    |   movel([0.279628, -1.417351, -2.542506, -0.752532, 1.570796, 1.850424],accel_mss,speed_ms,0,blend_radius_m)
    |   movel([0.279622, -1.416853, -2.542884, -0.752651, 1.570796, 1.850419],accel_mss,speed_ms,0,blend_radius_m)
    |   movel([0.279626, -1.416354, -2.543263, -0.752771, 1.570796, 1.850422],accel_mss,speed_ms,0,blend_radius_m)
    |   movel([0.279638, -1.416064, -2.543483, -0.752841, 1.570796, 1.850434],accel_mss,speed_ms,0,blend_radius_m)
    |   movel([0.279658, -1.415769, -2.543707, -0.752913, 1.570796, 1.850454],accel_mss,speed_ms,0,blend_radius_m)
    |   movel([0.279687, -1.415475, -2.543930, -0.752984, 1.570796, 1.850483],accel_mss,speed_ms,0,blend_radius_m)
    |   movel([0.279726, -1.415198, -2.544139, -0.753051, 1.570796, 1.850522],accel_mss,speed_ms,0,blend_radius_m)
    |   movel([0.279771, -1.414923, -2.544348, -0.753118, 1.570796, 1.850568],accel_mss,speed_ms,0,blend_radius_m)
    |   movel([0.279832, -1.414642, -2.544561, -0.753187, 1.570796, 1.850628],accel_mss,speed_ms,0,blend_radius_m)
    |   movel([0.279917, -1.414283, -2.544832, -0.753274, 1.570796, 1.850713],accel_mss,speed_ms,0,blend_radius_m)
    |   movel([0.280011, -1.413921, -2.545105, -0.753363, 1.570796, 1.850808],accel_mss,speed_ms,0,blend_radius_m)
    |   movel([0.280115, -1.413560, -2.545377, -0.753451, 1.570796, 1.850911],accel_mss,speed_ms,0,blend_radius_m)
    |   movel([0.280391, -1.412635, -2.546075, -0.753679, 1.570796, 1.851188],accel_mss,speed_ms,0,blend_radius_m)
    |   movel([0.280678, -1.411708, -2.546772, -0.753908, 1.570796, 1.851474],accel_mss,speed_ms,0,blend_radius_m)
    |   movel([0.280987, -1.410738, -2.547501, -0.754150, 1.570796, 1.851783],accel_mss,speed_ms,0,blend_radius_m)
    |   movel([0.281302, -1.409763, -2.548232, -0.754394, 1.570796, 1.852098],accel_mss,speed_ms,0,blend_radius_m)
    |   movel([0.281425, -1.409404, -2.548501, -0.754484, 1.570796, 1.852222],accel_mss,speed_ms,0,blend_radius_m)
    |   movel([0.281559, -1.409042, -2.548772, -0.754575, 1.570796, 1.852355],accel_mss,speed_ms,0,blend_radius_m)
    |   movel([0.281701, -1.408680, -2.549042, -0.754667, 1.570796, 1.852497],accel_mss,speed_ms,0,blend_radius_m)
    |   movel([0.281827, -1.408385, -2.549263, -0.754741, 1.570796, 1.852623],accel_mss,speed_ms,0,blend_radius_m)
    |   movel([0.281964, -1.408090, -2.549483, -0.754816, 1.570796, 1.852760],accel_mss,speed_ms,0,blend_radius_m)
    |   movel([0.282113, -1.407794, -2.549704, -0.754891, 1.570796, 1.852909],accel_mss,speed_ms,0,blend_radius_m)
    |   movel([0.282407, -1.407251, -2.550109, -0.755029, 1.570796, 1.853203],accel_mss,speed_ms,0,blend_radius_m)
    |   movel([0.282716, -1.406709, -2.550513, -0.755167, 1.570796, 1.853512],accel_mss,speed_ms,0,blend_radius_m)
    |   movel([0.283060, -1.406138, -2.550938, -0.755314, 1.570796, 1.853856],accel_mss,speed_ms,0,blend_radius_m)
    |   movel([0.283416, -1.405569, -2.551360, -0.755460, 1.570796, 1.854213],accel_mss,speed_ms,0,blend_radius_m)
    |   movel([0.283790, -1.405004, -2.551780, -0.755605, 1.570796, 1.854586],accel_mss,speed_ms,0,blend_radius_m)
    |   movel([0.284177, -1.404442, -2.552197, -0.755751, 1.570796, 1.854973],accel_mss,speed_ms,0,blend_radius_m)
    |   movel([0.284577, -1.403881, -2.552612, -0.755896, 1.570796, 1.855373],accel_mss,speed_ms,0,blend_radius_m)
    |   movel([0.284991, -1.403328, -2.553021, -0.756040, 1.570796, 1.855787],accel_mss,speed_ms,0,blend_radius_m)
    |   movel([0.285421, -1.402776, -2.553429, -0.756184, 1.570796, 1.856217],accel_mss,speed_ms,0,blend_radius_m)
    |   movel([0.285863, -1.402229, -2.553833, -0.756327, 1.570796, 1.856659],accel_mss,speed_ms,0,blend_radius_m)
    |   movel([0.286317, -1.401689, -2.554231, -0.756469, 1.570796, 1.857113],accel_mss,speed_ms,0,blend_radius_m)
    |   movel([0.286768, -1.401172, -2.554612, -0.756605, 1.570796, 1.857565],accel_mss,speed_ms,0,blend_radius_m)
    |   movel([0.287233, -1.400663, -2.554986, -0.756739, 1.570796, 1.858030],accel_mss,speed_ms,0,blend_radius_m)
    |   movel([0.287711, -1.400160, -2.555357, -0.756873, 1.570796, 1.858507],accel_mss,speed_ms,0,blend_radius_m)
    |   movel([0.288202, -1.399665, -2.555720, -0.757004, 1.570796, 1.858998],accel_mss,speed_ms,0,blend_radius_m)
    |   movel([0.288701, -1.399180, -2.556076, -0.757133, 1.570796, 1.859498],accel_mss,speed_ms,0,blend_radius_m)
    |   movel([0.289215, -1.398701, -2.556427, -0.757261, 1.570796, 1.860011],accel_mss,speed_ms,0,blend_radius_m)
    |   movel([0.289741, -1.398229, -2.556773, -0.757387, 1.570796, 1.860537],accel_mss,speed_ms,0,blend_radius_m)
    |   movel([0.290274, -1.397769, -2.557109, -0.757511, 1.570796, 1.861071],accel_mss,speed_ms,0,blend_radius_m)
    |   movel([0.290819, -1.397318, -2.557439, -0.757632, 1.570796, 1.861615],accel_mss,speed_ms,0,blend_radius_m)
    |   movel([0.291362, -1.396889, -2.557752, -0.757748, 1.570796, 1.862158],accel_mss,speed_ms,0,blend_radius_m)
    |   movel([0.291912, -1.396467, -2.558060, -0.757862, 1.570796, 1.862708],accel_mss,speed_ms,0,blend_radius_m)
    |   movel([0.292474, -1.396059, -2.558358, -0.757972, 1.570796, 1.863270],accel_mss,speed_ms,0,blend_radius_m)
    |   movel([0.293042, -1.395660, -2.558648, -0.758080, 1.570796, 1.863838],accel_mss,speed_ms,0,blend_radius_m)
    |   movel([0.293615, -1.395276, -2.558928, -0.758185, 1.570796, 1.864411],accel_mss,speed_ms,0,blend_radius_m)
    |   movel([0.294199, -1.394901, -2.559200, -0.758287, 1.570796, 1.864995],accel_mss,speed_ms,0,blend_radius_m)
    |   movel([0.294788, -1.394541, -2.559462, -0.758385, 1.570796, 1.865584],accel_mss,speed_ms,0,blend_radius_m)
    |   movel([0.295381, -1.394196, -2.559713, -0.758480, 1.570796, 1.866177],accel_mss,speed_ms,0,blend_radius_m)
    |   movel([0.295981, -1.393860, -2.559957, -0.758572, 1.570796, 1.866777],accel_mss,speed_ms,0,blend_radius_m)
    |   movel([0.296585, -1.393541, -2.560188, -0.758660, 1.570796, 1.867381],accel_mss,speed_ms,0,blend_radius_m)
    |   movel([0.297191, -1.393235, -2.560410, -0.758744, 1.570796, 1.867988],accel_mss,speed_ms,0,blend_radius_m)
    |   movel([0.297803, -1.392943, -2.560622, -0.758824, 1.570796, 1.868599],accel_mss,speed_ms,0,blend_radius_m)
    |   movel([0.298417, -1.392666, -2.560822, -0.758901, 1.570796, 1.869213],accel_mss,speed_ms,0,blend_radius_m)
    |   movel([0.299033, -1.392405, -2.561012, -0.758973, 1.570796, 1.869829],accel_mss,speed_ms,0,blend_radius_m)
    |   movel([0.299650, -1.392160, -2.561188, -0.759041, 1.570796, 1.870446],accel_mss,speed_ms,0,blend_radius_m)
    |   movel([0.300268, -1.391928, -2.561356, -0.759105, 1.570796, 1.871064],accel_mss,speed_ms,0,blend_radius_m)
    |   movel([0.300887, -1.391714, -2.561511, -0.759164, 1.570796, 1.871684],accel_mss,speed_ms,0,blend_radius_m)
    |   movel([0.301504, -1.391515, -2.561655, -0.759219, 1.570796, 1.872301],accel_mss,speed_ms,0,blend_radius_m)
    |   movel([0.302008, -1.391368, -2.561761, -0.759260, 1.570796, 1.872804],accel_mss,speed_ms,0,blend_radius_m)
    |   movel([0.302511, -1.391237, -2.561856, -0.759297, 1.570796, 1.873307],accel_mss,speed_ms,0,blend_radius_m)
    |   movel([0.303009, -1.391121, -2.561939, -0.759329, 1.570796, 1.873805],accel_mss,speed_ms,0,blend_radius_m)
    |   movel([0.303506, -1.391023, -2.562010, -0.759356, 1.570796, 1.874302],accel_mss,speed_ms,0,blend_radius_m)
    |   movel([0.304074, -1.390924, -2.562081, -0.759384, 1.570796, 1.874870],accel_mss,speed_ms,0,blend_radius_m)
    |   movel([0.304640, -1.390839, -2.562142, -0.759407, 1.570796, 1.875436],accel_mss,speed_ms,0,blend_radius_m)
    |   movel([0.305199, -1.390768, -2.562194, -0.759427, 1.570796, 1.875995],accel_mss,speed_ms,0,blend_radius_m)
    |   movel([0.305757, -1.390708, -2.562237, -0.759444, 1.570796, 1.876553],accel_mss,speed_ms,0,blend_radius_m)
    |   movel([0.306310, -1.390661, -2.562271, -0.759457, 1.570796, 1.877106],accel_mss,speed_ms,0,blend_radius_m)
    |   movel([0.306859, -1.390626, -2.562296, -0.759467, 1.570796, 1.877656],accel_mss,speed_ms,0,blend_radius_m)
    |   movel([0.307404, -1.390604, -2.562312, -0.759473, 1.570796, 1.878200],accel_mss,speed_ms,0,blend_radius_m)
    |   movel([0.307942, -1.390597, -2.562317, -0.759475, 1.570796, 1.878738],accel_mss,speed_ms,0,blend_radius_m)
    |   movel([0.308401, -1.390603, -2.562313, -0.759473, 1.570796, 1.879198],accel_mss,speed_ms,0,blend_radius_m)
    |   movel([0.308855, -1.390628, -2.562295, -0.759466, 1.570796, 1.879651],accel_mss,speed_ms,0,blend_radius_m)
    |   movel([0.309299, -1.390668, -2.562266, -0.759455, 1.570796, 1.880095],accel_mss,speed_ms,0,blend_radius_m)
    |   movel([0.309734, -1.390725, -2.562225, -0.759439, 1.570796, 1.880531],accel_mss,speed_ms,0,blend_radius_m)
    |   movel([0.310264, -1.390816, -2.562159, -0.759414, 1.570796, 1.881060],accel_mss,speed_ms,0,blend_radius_m)
    |   movel([0.310782, -1.390924, -2.562081, -0.759384, 1.570796, 1.881579],accel_mss,speed_ms,0,blend_radius_m)
    |   movel([0.311288, -1.391050, -2.561990, -0.759349, 1.570796, 1.882084],accel_mss,speed_ms,0,blend_radius_m)
    |   movel([0.311782, -1.391195, -2.561885, -0.759308, 1.570796, 1.882578],accel_mss,speed_ms,0,blend_radius_m)
    |   movel([0.312265, -1.391354, -2.561771, -0.759264, 1.570796, 1.883061],accel_mss,speed_ms,0,blend_radius_m)
    |   movel([0.312730, -1.391535, -2.561640, -0.759214, 1.570796, 1.883527],accel_mss,speed_ms,0,blend_radius_m)
    |   movel([0.313189, -1.391729, -2.561500, -0.759160, 1.570796, 1.883985],accel_mss,speed_ms,0,blend_radius_m)
    |   movel([0.313630, -1.391942, -2.561346, -0.759101, 1.570796, 1.884426],accel_mss,speed_ms,0,blend_radius_m)
    |   movel([0.314058, -1.392169, -2.561182, -0.759038, 1.570796, 1.884854],accel_mss,speed_ms,0,blend_radius_m)
    |   movel([0.314471, -1.392415, -2.561004, -0.758970, 1.570796, 1.885267],accel_mss,speed_ms,0,blend_radius_m)
    |   movel([0.314869, -1.392675, -2.560816, -0.758898, 1.570796, 1.885665],accel_mss,speed_ms,0,blend_radius_m)
    |   movel([0.315252, -1.392952, -2.560615, -0.758822, 1.570796, 1.886049],accel_mss,speed_ms,0,blend_radius_m)
    |   movel([0.315618, -1.393246, -2.560403, -0.758741, 1.570796, 1.886415],accel_mss,speed_ms,0,blend_radius_m)
    |   movel([0.315972, -1.393553, -2.560180, -0.758656, 1.570796, 1.886768],accel_mss,speed_ms,0,blend_radius_m)
    |   movel([0.316307, -1.393875, -2.559946, -0.758568, 1.570796, 1.887103],accel_mss,speed_ms,0,blend_radius_m)
    |   movel([0.316625, -1.394212, -2.559702, -0.758476, 1.570796, 1.887421],accel_mss,speed_ms,0,blend_radius_m)
    |   movel([0.316927, -1.394562, -2.559447, -0.758380, 1.570796, 1.887723],accel_mss,speed_ms,0,blend_radius_m)
    |   movel([0.317209, -1.394927, -2.559182, -0.758280, 1.570796, 1.888006],accel_mss,speed_ms,0,blend_radius_m)
    |   movel([0.317478, -1.395307, -2.558906, -0.758177, 1.570796, 1.888274],accel_mss,speed_ms,0,blend_radius_m)
    |   movel([0.317727, -1.395700, -2.558619, -0.758070, 1.570796, 1.888523],accel_mss,speed_ms,0,blend_radius_m)
    |   movel([0.317959, -1.396104, -2.558325, -0.757960, 1.570796, 1.888756],accel_mss,speed_ms,0,blend_radius_m)
    |   movel([0.318170, -1.396522, -2.558020, -0.757847, 1.570796, 1.888966],accel_mss,speed_ms,0,blend_radius_m)
    |   movel([0.318366, -1.396949, -2.557708, -0.757731, 1.570796, 1.889162],accel_mss,speed_ms,0,blend_radius_m)
    |   movel([0.318541, -1.397389, -2.557387, -0.757613, 1.570796, 1.889338],accel_mss,speed_ms,0,blend_radius_m)
    |   movel([0.318684, -1.397780, -2.557101, -0.757508, 1.570796, 1.889480],accel_mss,speed_ms,0,blend_radius_m)
    |   movel([0.318813, -1.398180, -2.556808, -0.757400, 1.570796, 1.889610],accel_mss,speed_ms,0,blend_radius_m)
    |   movel([0.318930, -1.398586, -2.556511, -0.757292, 1.570796, 1.889726],accel_mss,speed_ms,0,blend_radius_m)
    |   movel([0.319035, -1.398997, -2.556210, -0.757182, 1.570796, 1.889832],accel_mss,speed_ms,0,blend_radius_m)
    |   movel([0.319122, -1.399383, -2.555927, -0.757079, 1.570796, 1.889918],accel_mss,speed_ms,0,blend_radius_m)
    |   movel([0.319192, -1.399776, -2.555638, -0.756974, 1.570796, 1.889989],accel_mss,speed_ms,0,blend_radius_m)
    |   movel([0.319252, -1.400175, -2.555345, -0.756868, 1.570796, 1.890048],accel_mss,speed_ms,0,blend_radius_m)
    |   movel([0.319295, -1.400581, -2.555047, -0.756761, 1.570796, 1.890091],accel_mss,speed_ms,0,blend_radius_m)
    |   movel([0.319326, -1.401001, -2.554738, -0.756650, 1.570796, 1.890123],accel_mss,speed_ms,0,blend_radius_m)
    |   movel([0.319344, -1.401428, -2.554424, -0.756537, 1.570796, 1.890140],accel_mss,speed_ms,0,blend_radius_m)
    |   movel([0.319347, -1.401858, -2.554107, -0.756424, 1.570796, 1.890143],accel_mss,speed_ms,0,blend_radius_m)
    |   movel([0.319338, -1.402295, -2.553784, -0.756310, 1.570796, 1.890134],accel_mss,speed_ms,0,blend_radius_m)
    |   movel([0.319303, -1.402955, -2.553297, -0.756137, 1.570796, 1.890099],accel_mss,speed_ms,0,blend_radius_m)
    |   movel([0.319250, -1.403620, -2.552805, -0.755964, 1.570796, 1.890046],accel_mss,speed_ms,0,blend_radius_m)
    |   movel([0.319177, -1.404290, -2.552309, -0.755790, 1.570796, 1.889973],accel_mss,speed_ms,0,blend_radius_m)
    |   movel([0.319122, -1.404672, -2.552026, -0.755691, 1.570796, 1.889918],accel_mss,speed_ms,0,blend_radius_m)
    |   movel([0.319055, -1.405054, -2.551743, -0.755592, 1.570796, 1.889852],accel_mss,speed_ms,0,blend_radius_m)
    |   movel([0.318973, -1.405442, -2.551455, -0.755492, 1.570796, 1.889770],accel_mss,speed_ms,0,blend_radius_m)
    |   movel([0.318880, -1.405830, -2.551166, -0.755393, 1.570796, 1.889676],accel_mss,speed_ms,0,blend_radius_m)
    |   movel([0.318769, -1.406222, -2.550875, -0.755292, 1.570796, 1.889566],accel_mss,speed_ms,0,blend_radius_m)
    |   movel([0.318582, -1.406841, -2.550414, -0.755134, 1.570796, 1.889378],accel_mss,speed_ms,0,blend_radius_m)
    |   movel([0.318379, -1.407463, -2.549951, -0.754975, 1.570796, 1.889176],accel_mss,speed_ms,0,blend_radius_m)
    |   movel([0.318164, -1.408086, -2.549486, -0.754817, 1.570796, 1.888960],accel_mss,speed_ms,0,blend_radius_m)
    |   movel([0.317935, -1.408706, -2.549023, -0.754660, 1.570796, 1.888732],accel_mss,speed_ms,0,blend_radius_m)
    |   movel([0.317694, -1.409332, -2.548555, -0.754502, 1.570796, 1.888490],accel_mss,speed_ms,0,blend_radius_m)
    |   movel([0.317439, -1.409957, -2.548086, -0.754345, 1.570796, 1.888236],accel_mss,speed_ms,0,blend_radius_m)
    |   movel([0.317172, -1.410581, -2.547619, -0.754189, 1.570796, 1.887968],accel_mss,speed_ms,0,blend_radius_m)
    |   movel([0.316891, -1.411206, -2.547150, -0.754033, 1.570796, 1.887688],accel_mss,speed_ms,0,blend_radius_m)
    |   movel([0.316702, -1.411607, -2.546849, -0.753934, 1.570796, 1.887499],accel_mss,speed_ms,0,blend_radius_m)
    |   movel([0.316500, -1.412006, -2.546548, -0.753834, 1.570796, 1.887297],accel_mss,speed_ms,0,blend_radius_m)
    |   movel([0.316286, -1.412404, -2.546249, -0.753736, 1.570796, 1.887082],accel_mss,speed_ms,0,blend_radius_m)
    |   movel([0.316060, -1.412801, -2.545950, -0.753638, 1.570796, 1.886857],accel_mss,speed_ms,0,blend_radius_m)
    |   movel([0.315822, -1.413196, -2.545652, -0.753541, 1.570796, 1.886618],accel_mss,speed_ms,0,blend_radius_m)
    |   movel([0.315491, -1.413724, -2.545254, -0.753411, 1.570796, 1.886288],accel_mss,speed_ms,0,blend_radius_m)
    |   movel([0.315149, -1.414246, -2.544860, -0.753283, 1.570796, 1.885946],accel_mss,speed_ms,0,blend_radius_m)
    |   movel([0.314795, -1.414766, -2.544466, -0.753156, 1.570796, 1.885591],accel_mss,speed_ms,0,blend_radius_m)
    |   movel([0.314428, -1.415283, -2.544075, -0.753031, 1.570796, 1.885224],accel_mss,speed_ms,0,blend_radius_m)
    |   movel([0.314052, -1.415796, -2.543687, -0.752906, 1.570796, 1.884848],accel_mss,speed_ms,0,blend_radius_m)
    |   speed_ms = 0.003
    |   movel([0.314052, -1.418980, -2.545116, -0.748292, 1.570796, 1.884848],accel_mss,speed_ms,0,blend_radius_m)
    |   speed_ms = 0.007
    |   movel([0.313677, -1.419471, -2.544743, -0.748176, 1.570796, 1.884473],accel_mss,speed_ms,0,blend_radius_m)
    |   movel([0.313291, -1.419955, -2.544373, -0.748061, 1.570796, 1.884087],accel_mss,speed_ms,0,blend_radius_m)
    |   movel([0.312894, -1.420434, -2.544007, -0.747947, 1.570796, 1.883690],accel_mss,speed_ms,0,blend_radius_m)
    |   movel([0.312488, -1.420907, -2.543646, -0.747836, 1.570796, 1.883284],accel_mss,speed_ms,0,blend_radius_m)
    |   movel([0.312070, -1.421375, -2.543288, -0.747726, 1.570796, 1.882867],accel_mss,speed_ms,0,blend_radius_m)
    |   movel([0.311650, -1.421828, -2.542941, -0.747620, 1.570796, 1.882446],accel_mss,speed_ms,0,blend_radius_m)
    |   movel([0.311220, -1.422275, -2.542599, -0.747515, 1.570796, 1.882017],accel_mss,speed_ms,0,blend_radius_m)
    |   movel([0.310783, -1.422715, -2.542262, -0.747413, 1.570796, 1.881579],accel_mss,speed_ms,0,blend_radius_m)
    |   movel([0.310335, -1.423146, -2.541930, -0.747312, 1.570796, 1.881131],accel_mss,speed_ms,0,blend_radius_m)
    |   movel([0.309878, -1.423572, -2.541603, -0.747214, 1.570796, 1.880674],accel_mss,speed_ms,0,blend_radius_m)
    |   movel([0.309414, -1.423989, -2.541283, -0.747117, 1.570796, 1.880210],accel_mss,speed_ms,0,blend_radius_m)
    |   movel([0.308942, -1.424397, -2.540969, -0.747023, 1.570796, 1.879738],accel_mss,speed_ms,0,blend_radius_m)
    |   movel([0.308461, -1.424798, -2.540660, -0.746931, 1.570796, 1.879258],accel_mss,speed_ms,0,blend_radius_m)
    |   movel([0.307976, -1.425188, -2.540359, -0.746842, 1.570796, 1.878772],accel_mss,speed_ms,0,blend_radius_m)
    |   movel([0.307480, -1.425572, -2.540063, -0.746754, 1.570796, 1.878276],accel_mss,speed_ms,0,blend_radius_m)
    |   movel([0.307008, -1.425924, -2.539791, -0.746674, 1.570796, 1.877805],accel_mss,speed_ms,0,blend_radius_m)
    |   movel([0.306532, -1.426271, -2.539524, -0.746595, 1.570796, 1.877329],accel_mss,speed_ms,0,blend_radius_m)
    |   movel([0.306049, -1.426607, -2.539263, -0.746518, 1.570796, 1.876845],accel_mss,speed_ms,0,blend_radius_m)
    |   movel([0.305564, -1.426936, -2.539009, -0.746444, 1.570796, 1.876360],accel_mss,speed_ms,0,blend_radius_m)
    |   movel([0.305072, -1.427259, -2.538759, -0.746371, 1.570796, 1.875869],accel_mss,speed_ms,0,blend_radius_m)
    |   movel([0.304596, -1.427558, -2.538528, -0.746303, 1.570796, 1.875392],accel_mss,speed_ms,0,blend_radius_m)
    |   movel([0.304118, -1.427847, -2.538304, -0.746238, 1.570796, 1.874915],accel_mss,speed_ms,0,blend_radius_m)
    |   movel([0.303635, -1.428129, -2.538085, -0.746175, 1.570796, 1.874431],accel_mss,speed_ms,0,blend_radius_m)
    |   movel([0.303149, -1.428400, -2.537875, -0.746114, 1.570796, 1.873945],accel_mss,speed_ms,0,blend_radius_m)
    |   movel([0.302659, -1.428662, -2.537672, -0.746055, 1.570796, 1.873456],accel_mss,speed_ms,0,blend_radius_m)
    |   movel([0.302165, -1.428914, -2.537476, -0.745999, 1.570796, 1.872961],accel_mss,speed_ms,0,blend_radius_m)
    |   movel([0.301669, -1.429155, -2.537289, -0.745945, 1.570796, 1.872465],accel_mss,speed_ms,0,blend_radius_m)
    |   movel([0.301171, -1.429387, -2.537108, -0.745893, 1.570796, 1.871967],accel_mss,speed_ms,0,blend_radius_m)
    |   movel([0.300669, -1.429609, -2.536936, -0.745844, 1.570796, 1.871465],accel_mss,speed_ms,0,blend_radius_m)
    |   movel([0.300169, -1.429819, -2.536773, -0.745797, 1.570796, 1.870966],accel_mss,speed_ms,0,blend_radius_m)
    |   movel([0.299643, -1.430029, -2.536609, -0.745751, 1.570796, 1.870440],accel_mss,speed_ms,0,blend_radius_m)
    |   movel([0.299116, -1.430229, -2.536454, -0.745706, 1.570796, 1.869913],accel_mss,speed_ms,0,blend_radius_m)
    |   movel([0.298589, -1.430419, -2.536306, -0.745664, 1.570796, 1.869385],accel_mss,speed_ms,0,blend_radius_m)
    |   movel([0.298060, -1.430599, -2.536165, -0.745625, 1.570796, 1.868856],accel_mss,speed_ms,0,blend_radius_m)
    |   movel([0.297533, -1.430769, -2.536033, -0.745587, 1.570796, 1.868329],accel_mss,speed_ms,0,blend_radius_m)
    |   movel([0.297159, -1.430881, -2.535946, -0.745562, 1.570796, 1.867955],accel_mss,speed_ms,0,blend_radius_m)
    |   movel([0.296785, -1.430981, -2.535868, -0.745540, 1.570796, 1.867581],accel_mss,speed_ms,0,blend_radius_m)
    |   movel([0.296415, -1.431068, -2.535800, -0.745521, 1.570796, 1.867211],accel_mss,speed_ms,0,blend_radius_m)
    |   movel([0.296044, -1.431146, -2.535739, -0.745504, 1.570796, 1.866840],accel_mss,speed_ms,0,blend_radius_m)
    |   movel([0.295677, -1.431211, -2.535688, -0.745490, 1.570796, 1.866474],accel_mss,speed_ms,0,blend_radius_m)
    |   movel([0.295078, -1.431301, -2.535618, -0.745470, 1.570796, 1.865874],accel_mss,speed_ms,0,blend_radius_m)
    |   movel([0.294481, -1.431382, -2.535555, -0.745452, 1.570796, 1.865278],accel_mss,speed_ms,0,blend_radius_m)
    |   movel([0.293889, -1.431452, -2.535500, -0.745437, 1.570796, 1.864685],accel_mss,speed_ms,0,blend_radius_m)
    |   movel([0.293298, -1.431509, -2.535456, -0.745424, 1.570796, 1.864095],accel_mss,speed_ms,0,blend_radius_m)
    |   movel([0.292712, -1.431558, -2.535417, -0.745413, 1.570796, 1.863509],accel_mss,speed_ms,0,blend_radius_m)
    |   movel([0.292131, -1.431595, -2.535388, -0.745405, 1.570796, 1.862927],accel_mss,speed_ms,0,blend_radius_m)
    |   movel([0.291553, -1.431620, -2.535369, -0.745400, 1.570796, 1.862349],accel_mss,speed_ms,0,blend_radius_m)
    |   movel([0.290978, -1.431636, -2.535356, -0.745396, 1.570796, 1.861774],accel_mss,speed_ms,0,blend_radius_m)
    |   movel([0.290633, -1.431636, -2.535357, -0.745396, 1.570796, 1.861429],accel_mss,speed_ms,0,blend_radius_m)
    |   movel([0.290291, -1.431623, -2.535367, -0.745399, 1.570796, 1.861088],accel_mss,speed_ms,0,blend_radius_m)
    |   movel([0.289956, -1.431600, -2.535385, -0.745404, 1.570796, 1.860752],accel_mss,speed_ms,0,blend_radius_m)
    |   movel([0.289629, -1.431563, -2.535413, -0.745412, 1.570796, 1.860425],accel_mss,speed_ms,0,blend_radius_m)
    |   movel([0.289306, -1.431515, -2.535451, -0.745423, 1.570796, 1.860102],accel_mss,speed_ms,0,blend_radius_m)
    |   movel([0.288849, -1.431430, -2.535517, -0.745442, 1.570796, 1.859645],accel_mss,speed_ms,0,blend_radius_m)
    |   movel([0.288400, -1.431335, -2.535592, -0.745462, 1.570796, 1.859196],accel_mss,speed_ms,0,blend_radius_m)
    |   movel([0.287956, -1.431229, -2.535674, -0.745486, 1.570796, 1.858752],accel_mss,speed_ms,0,blend_radius_m)
    |   movel([0.287522, -1.431112, -2.535765, -0.745511, 1.570796, 1.858319],accel_mss,speed_ms,0,blend_radius_m)
    |   movel([0.287095, -1.430983, -2.535866, -0.745540, 1.570796, 1.857891],accel_mss,speed_ms,0,blend_radius_m)
    |   movel([0.286701, -1.430853, -2.535968, -0.745569, 1.570796, 1.857497],accel_mss,speed_ms,0,blend_radius_m)
    |   movel([0.286315, -1.430708, -2.536081, -0.745601, 1.570796, 1.857112],accel_mss,speed_ms,0,blend_radius_m)
    |   movel([0.285940, -1.430552, -2.536202, -0.745635, 1.570796, 1.856736],accel_mss,speed_ms,0,blend_radius_m)
    |   movel([0.285575, -1.430384, -2.536333, -0.745672, 1.570796, 1.856371],accel_mss,speed_ms,0,blend_radius_m)
    |   movel([0.285220, -1.430204, -2.536473, -0.745712, 1.570796, 1.856016],accel_mss,speed_ms,0,blend_radius_m)
    |   movel([0.284876, -1.430011, -2.536623, -0.745755, 1.570796, 1.855672],accel_mss,speed_ms,0,blend_radius_m)
    |   movel([0.284542, -1.429806, -2.536782, -0.745800, 1.570796, 1.855338],accel_mss,speed_ms,0,blend_radius_m)
    |   movel([0.284217, -1.429591, -2.536950, -0.745848, 1.570796, 1.855014],accel_mss,speed_ms,0,blend_radius_m)
    |   movel([0.283905, -1.429364, -2.537126, -0.745898, 1.570796, 1.854702],accel_mss,speed_ms,0,blend_radius_m)
    |   movel([0.283606, -1.429126, -2.537311, -0.745951, 1.570796, 1.854402],accel_mss,speed_ms,0,blend_radius_m)
    |   movel([0.283296, -1.428863, -2.537516, -0.746010, 1.570796, 1.854092],accel_mss,speed_ms,0,blend_radius_m)
    |   movel([0.282998, -1.428590, -2.537728, -0.746071, 1.570796, 1.853794],accel_mss,speed_ms,0,blend_radius_m)
    |   movel([0.282710, -1.428306, -2.537948, -0.746135, 1.570796, 1.853506],accel_mss,speed_ms,0,blend_radius_m)
    |   movel([0.282433, -1.428013, -2.538175, -0.746201, 1.570796, 1.853230],accel_mss,speed_ms,0,blend_radius_m)
    |   movel([0.282168, -1.427713, -2.538408, -0.746268, 1.570796, 1.852964],accel_mss,speed_ms,0,blend_radius_m)
    |   movel([0.281908, -1.427391, -2.538657, -0.746341, 1.570796, 1.852705],accel_mss,speed_ms,0,blend_radius_m)
    |   movel([0.281660, -1.427063, -2.538911, -0.746415, 1.570796, 1.852456],accel_mss,speed_ms,0,blend_radius_m)
    |   movel([0.281424, -1.426723, -2.539174, -0.746492, 1.570796, 1.852220],accel_mss,speed_ms,0,blend_radius_m)
    |   movel([0.281204, -1.426373, -2.539445, -0.746571, 1.570796, 1.852000],accel_mss,speed_ms,0,blend_radius_m)
    |   movel([0.280995, -1.426015, -2.539721, -0.746653, 1.570796, 1.851791],accel_mss,speed_ms,0,blend_radius_m)
    |   movel([0.280805, -1.425654, -2.540000, -0.746735, 1.570796, 1.851601],accel_mss,speed_ms,0,blend_radius_m)
    |   movel([0.280628, -1.425285, -2.540285, -0.746819, 1.570796, 1.851424],accel_mss,speed_ms,0,blend_radius_m)
    |   movel([0.280467, -1.424906, -2.540577, -0.746906, 1.570796, 1.851263],accel_mss,speed_ms,0,blend_radius_m)
    |   movel([0.280320, -1.424517, -2.540876, -0.746996, 1.570796, 1.851116],accel_mss,speed_ms,0,blend_radius_m)
    |   movel([0.280187, -1.424121, -2.541181, -0.747087, 1.570796, 1.850983],accel_mss,speed_ms,0,blend_radius_m)
    |   movel([0.280067, -1.423708, -2.541499, -0.747182, 1.570796, 1.850863],accel_mss,speed_ms,0,blend_radius_m)
    |   movel([0.279961, -1.423286, -2.541823, -0.747280, 1.570796, 1.850757],accel_mss,speed_ms,0,blend_radius_m)
    |   movel([0.279870, -1.422858, -2.542152, -0.747379, 1.570796, 1.850667],accel_mss,speed_ms,0,blend_radius_m)
    |   movel([0.279795, -1.422422, -2.542486, -0.747481, 1.570796, 1.850592],accel_mss,speed_ms,0,blend_radius_m)
    |   movel([0.279735, -1.421980, -2.542825, -0.747584, 1.570796, 1.850532],accel_mss,speed_ms,0,blend_radius_m)
    |   movel([0.279686, -1.421501, -2.543192, -0.747696, 1.570796, 1.850483],accel_mss,speed_ms,0,blend_radius_m)
    |   movel([0.279652, -1.421019, -2.543561, -0.747810, 1.570796, 1.850448],accel_mss,speed_ms,0,blend_radius_m)
    |   movel([0.279628, -1.420531, -2.543934, -0.747925, 1.570796, 1.850424],accel_mss,speed_ms,0,blend_radius_m)
    |   movel([0.279622, -1.420035, -2.544313, -0.748042, 1.570796, 1.850419],accel_mss,speed_ms,0,blend_radius_m)
    |   movel([0.279626, -1.419537, -2.544692, -0.748160, 1.570796, 1.850422],accel_mss,speed_ms,0,blend_radius_m)
    |   movel([0.279638, -1.419248, -2.544913, -0.748229, 1.570796, 1.850434],accel_mss,speed_ms,0,blend_radius_m)
    |   movel([0.279658, -1.418954, -2.545137, -0.748299, 1.570796, 1.850454],accel_mss,speed_ms,0,blend_radius_m)
    |   movel([0.279687, -1.418660, -2.545360, -0.748369, 1.570796, 1.850483],accel_mss,speed_ms,0,blend_radius_m)
    |   movel([0.279726, -1.418384, -2.545570, -0.748435, 1.570796, 1.850522],accel_mss,speed_ms,0,blend_radius_m)
    |   movel([0.279771, -1.418110, -2.545779, -0.748500, 1.570796, 1.850568],accel_mss,speed_ms,0,blend_radius_m)
    |   movel([0.279832, -1.417829, -2.545992, -0.748568, 1.570796, 1.850628],accel_mss,speed_ms,0,blend_radius_m)
    |   movel([0.279917, -1.417472, -2.546264, -0.748654, 1.570796, 1.850713],accel_mss,speed_ms,0,blend_radius_m)
    |   movel([0.280011, -1.417111, -2.546538, -0.748740, 1.570796, 1.850808],accel_mss,speed_ms,0,blend_radius_m)
    |   movel([0.280115, -1.416751, -2.546811, -0.748827, 1.570796, 1.850911],accel_mss,speed_ms,0,blend_radius_m)
    |   movel([0.280391, -1.415829, -2.547509, -0.749051, 1.570796, 1.851188],accel_mss,speed_ms,0,blend_radius_m)
    |   movel([0.280678, -1.414904, -2.548209, -0.749276, 1.570796, 1.851474],accel_mss,speed_ms,0,blend_radius_m)
    |   movel([0.280987, -1.413936, -2.548939, -0.749513, 1.570796, 1.851783],accel_mss,speed_ms,0,blend_radius_m)
    |   movel([0.281302, -1.412965, -2.549671, -0.749753, 1.570796, 1.852098],accel_mss,speed_ms,0,blend_radius_m)
    |   movel([0.281425, -1.412607, -2.549941, -0.749842, 1.570796, 1.852222],accel_mss,speed_ms,0,blend_radius_m)
    |   movel([0.281559, -1.412245, -2.550213, -0.749931, 1.570796, 1.852355],accel_mss,speed_ms,0,blend_radius_m)
    |   movel([0.281701, -1.411885, -2.550483, -0.750021, 1.570796, 1.852497],accel_mss,speed_ms,0,blend_radius_m)
    |   movel([0.281827, -1.411590, -2.550704, -0.750094, 1.570796, 1.852623],accel_mss,speed_ms,0,blend_radius_m)
    |   movel([0.281964, -1.411296, -2.550925, -0.750168, 1.570796, 1.852760],accel_mss,speed_ms,0,blend_radius_m)
    |   movel([0.282113, -1.411001, -2.551146, -0.750241, 1.570796, 1.852909],accel_mss,speed_ms,0,blend_radius_m)
    |   movel([0.282407, -1.410459, -2.551553, -0.750377, 1.570796, 1.853203],accel_mss,speed_ms,0,blend_radius_m)
    |   movel([0.282716, -1.409919, -2.551957, -0.750513, 1.570796, 1.853512],accel_mss,speed_ms,0,blend_radius_m)
    |   movel([0.283060, -1.409349, -2.552383, -0.750657, 1.570796, 1.853856],accel_mss,speed_ms,0,blend_radius_m)
    |   movel([0.283416, -1.408782, -2.552807, -0.750800, 1.570796, 1.854213],accel_mss,speed_ms,0,blend_radius_m)
    |   movel([0.283790, -1.408219, -2.553227, -0.750943, 1.570796, 1.854586],accel_mss,speed_ms,0,blend_radius_m)
    |   movel([0.284177, -1.407658, -2.553645, -0.751086, 1.570796, 1.854973],accel_mss,speed_ms,0,blend_radius_m)
    |   movel([0.284577, -1.407099, -2.554061, -0.751229, 1.570796, 1.855373],accel_mss,speed_ms,0,blend_radius_m)
    |   movel([0.284991, -1.406547, -2.554471, -0.751371, 1.570796, 1.855787],accel_mss,speed_ms,0,blend_radius_m)
    |   movel([0.285421, -1.405997, -2.554880, -0.751512, 1.570796, 1.856217],accel_mss,speed_ms,0,blend_radius_m)
    |   movel([0.285863, -1.405452, -2.555284, -0.751653, 1.570796, 1.856659],accel_mss,speed_ms,0,blend_radius_m)
    |   movel([0.286317, -1.404913, -2.555684, -0.751792, 1.570796, 1.857113],accel_mss,speed_ms,0,blend_radius_m)
    |   movel([0.286768, -1.404397, -2.556065, -0.751926, 1.570796, 1.857565],accel_mss,speed_ms,0,blend_radius_m)
    |   movel([0.287233, -1.403890, -2.556440, -0.752058, 1.570796, 1.858030],accel_mss,speed_ms,0,blend_radius_m)
    |   movel([0.287711, -1.403388, -2.556811, -0.752189, 1.570796, 1.858507],accel_mss,speed_ms,0,blend_radius_m)
    |   movel([0.288202, -1.402895, -2.557176, -0.752319, 1.570796, 1.858998],accel_mss,speed_ms,0,blend_radius_m)
    |   movel([0.288701, -1.402411, -2.557533, -0.752446, 1.570796, 1.859498],accel_mss,speed_ms,0,blend_radius_m)
    |   movel([0.289215, -1.401933, -2.557884, -0.752571, 1.570796, 1.860011],accel_mss,speed_ms,0,blend_radius_m)
    |   movel([0.289741, -1.401463, -2.558231, -0.752696, 1.570796, 1.860537],accel_mss,speed_ms,0,blend_radius_m)
    |   movel([0.290274, -1.401004, -2.558568, -0.752817, 1.570796, 1.861071],accel_mss,speed_ms,0,blend_radius_m)
    |   movel([0.290819, -1.400554, -2.558898, -0.752936, 1.570796, 1.861615],accel_mss,speed_ms,0,blend_radius_m)
    |   movel([0.291362, -1.400126, -2.559213, -0.753050, 1.570796, 1.862158],accel_mss,speed_ms,0,blend_radius_m)
    |   movel([0.291912, -1.399705, -2.559521, -0.753162, 1.570796, 1.862708],accel_mss,speed_ms,0,blend_radius_m)
    |   movel([0.292474, -1.399298, -2.559820, -0.753271, 1.570796, 1.863270],accel_mss,speed_ms,0,blend_radius_m)
    |   movel([0.293042, -1.398901, -2.560111, -0.753378, 1.570796, 1.863838],accel_mss,speed_ms,0,blend_radius_m)
    |   movel([0.293615, -1.398518, -2.560391, -0.753480, 1.570796, 1.864411],accel_mss,speed_ms,0,blend_radius_m)
    |   movel([0.294199, -1.398144, -2.560664, -0.753581, 1.570796, 1.864995],accel_mss,speed_ms,0,blend_radius_m)
    |   movel([0.294788, -1.397785, -2.560926, -0.753678, 1.570796, 1.865584],accel_mss,speed_ms,0,blend_radius_m)
    |   movel([0.295381, -1.397440, -2.561178, -0.753771, 1.570796, 1.866177],accel_mss,speed_ms,0,blend_radius_m)
    |   movel([0.295981, -1.397106, -2.561422, -0.753861, 1.570796, 1.866777],accel_mss,speed_ms,0,blend_radius_m)
    |   movel([0.296585, -1.396788, -2.561654, -0.753947, 1.570796, 1.867381],accel_mss,speed_ms,0,blend_radius_m)
    |   movel([0.297191, -1.396482, -2.561876, -0.754030, 1.570796, 1.867988],accel_mss,speed_ms,0,blend_radius_m)
    |   movel([0.297803, -1.396191, -2.562088, -0.754109, 1.570796, 1.868599],accel_mss,speed_ms,0,blend_radius_m)
    |   movel([0.298417, -1.395915, -2.562289, -0.754184, 1.570796, 1.869213],accel_mss,speed_ms,0,blend_radius_m)
    |   movel([0.299033, -1.395654, -2.562479, -0.754256, 1.570796, 1.869829],accel_mss,speed_ms,0,blend_radius_m)
    |   movel([0.299650, -1.395410, -2.562656, -0.754322, 1.570796, 1.870446],accel_mss,speed_ms,0,blend_radius_m)
    |   movel([0.300268, -1.395179, -2.562824, -0.754385, 1.570796, 1.871064],accel_mss,speed_ms,0,blend_radius_m)
    |   movel([0.300887, -1.394965, -2.562980, -0.754444, 1.570796, 1.871684],accel_mss,speed_ms,0,blend_radius_m)
    |   movel([0.301504, -1.394767, -2.563124, -0.754498, 1.570796, 1.872301],accel_mss,speed_ms,0,blend_radius_m)
    |   movel([0.302008, -1.394621, -2.563230, -0.754538, 1.570796, 1.872804],accel_mss,speed_ms,0,blend_radius_m)
    |   movel([0.302511, -1.394490, -2.563325, -0.754574, 1.570796, 1.873307],accel_mss,speed_ms,0,blend_radius_m)
    |   movel([0.303009, -1.394374, -2.563409, -0.754606, 1.570796, 1.873805],accel_mss,speed_ms,0,blend_radius_m)
    |   movel([0.303506, -1.394276, -2.563480, -0.754633, 1.570796, 1.874302],accel_mss,speed_ms,0,blend_radius_m)
    |   movel([0.304074, -1.394178, -2.563551, -0.754660, 1.570796, 1.874870],accel_mss,speed_ms,0,blend_radius_m)
    |   movel([0.304640, -1.394093, -2.563612, -0.754683, 1.570796, 1.875436],accel_mss,speed_ms,0,blend_radius_m)
    |   movel([0.305199, -1.394022, -2.563664, -0.754703, 1.570796, 1.875995],accel_mss,speed_ms,0,blend_radius_m)
    |   movel([0.305757, -1.393962, -2.563707, -0.754720, 1.570796, 1.876553],accel_mss,speed_ms,0,blend_radius_m)
    |   movel([0.306310, -1.393916, -2.563741, -0.754732, 1.570796, 1.877106],accel_mss,speed_ms,0,blend_radius_m)
    |   movel([0.306859, -1.393881, -2.563766, -0.754742, 1.570796, 1.877656],accel_mss,speed_ms,0,blend_radius_m)
    |   movel([0.307404, -1.393859, -2.563782, -0.754748, 1.570796, 1.878200],accel_mss,speed_ms,0,blend_radius_m)
    |   movel([0.307942, -1.393852, -2.563787, -0.754750, 1.570796, 1.878738],accel_mss,speed_ms,0,blend_radius_m)
    |   movel([0.308401, -1.393858, -2.563783, -0.754748, 1.570796, 1.879198],accel_mss,speed_ms,0,blend_radius_m)
    |   movel([0.308855, -1.393882, -2.563765, -0.754741, 1.570796, 1.879651],accel_mss,speed_ms,0,blend_radius_m)
    |   movel([0.309299, -1.393923, -2.563736, -0.754730, 1.570796, 1.880095],accel_mss,speed_ms,0,blend_radius_m)
    |   movel([0.309734, -1.393979, -2.563695, -0.754715, 1.570796, 1.880531],accel_mss,speed_ms,0,blend_radius_m)
    |   movel([0.310264, -1.394070, -2.563629, -0.754690, 1.570796, 1.881060],accel_mss,speed_ms,0,blend_radius_m)
    |   movel([0.310782, -1.394178, -2.563551, -0.754660, 1.570796, 1.881579],accel_mss,speed_ms,0,blend_radius_m)
    |   movel([0.311288, -1.394304, -2.563460, -0.754626, 1.570796, 1.882084],accel_mss,speed_ms,0,blend_radius_m)
    |   movel([0.311782, -1.394448, -2.563355, -0.754586, 1.570796, 1.882578],accel_mss,speed_ms,0,blend_radius_m)
    |   movel([0.312265, -1.394607, -2.563240, -0.754542, 1.570796, 1.883061],accel_mss,speed_ms,0,blend_radius_m)
    |   movel([0.312730, -1.394787, -2.563109, -0.754493, 1.570796, 1.883527],accel_mss,speed_ms,0,blend_radius_m)
    |   movel([0.313189, -1.394980, -2.562969, -0.754440, 1.570796, 1.883985],accel_mss,speed_ms,0,blend_radius_m)
    |   movel([0.313630, -1.395193, -2.562814, -0.754382, 1.570796, 1.884426],accel_mss,speed_ms,0,blend_radius_m)
    |   movel([0.314058, -1.395419, -2.562650, -0.754320, 1.570796, 1.884854],accel_mss,speed_ms,0,blend_radius_m)
    |   movel([0.314471, -1.395665, -2.562471, -0.754253, 1.570796, 1.885267],accel_mss,speed_ms,0,blend_radius_m)
    |   movel([0.314869, -1.395924, -2.562283, -0.754182, 1.570796, 1.885665],accel_mss,speed_ms,0,blend_radius_m)
    |   movel([0.315252, -1.396200, -2.562082, -0.754107, 1.570796, 1.886049],accel_mss,speed_ms,0,blend_radius_m)
    |   movel([0.315618, -1.396493, -2.561869, -0.754027, 1.570796, 1.886415],accel_mss,speed_ms,0,blend_radius_m)
    |   movel([0.315972, -1.396800, -2.561645, -0.753944, 1.570796, 1.886768],accel_mss,speed_ms,0,blend_radius_m)
    |   movel([0.316307, -1.397121, -2.561411, -0.753857, 1.570796, 1.887103],accel_mss,speed_ms,0,blend_radius_m)
    |   movel([0.316625, -1.397456, -2.561166, -0.753766, 1.570796, 1.887421],accel_mss,speed_ms,0,blend_radius_m)
    |   movel([0.316927, -1.397806, -2.560911, -0.753672, 1.570796, 1.887723],accel_mss,speed_ms,0,blend_radius_m)
    |   movel([0.317209, -1.398170, -2.560645, -0.753574, 1.570796, 1.888006],accel_mss,speed_ms,0,blend_radius_m)
    |   movel([0.317478, -1.398548, -2.560368, -0.753472, 1.570796, 1.888274],accel_mss,speed_ms,0,blend_radius_m)
    |   movel([0.317727, -1.398941, -2.560081, -0.753367, 1.570796, 1.888523],accel_mss,speed_ms,0,blend_radius_m)
    |   movel([0.317959, -1.399343, -2.559787, -0.753259, 1.570796, 1.888756],accel_mss,speed_ms,0,blend_radius_m)
    |   movel([0.318170, -1.399760, -2.559481, -0.753148, 1.570796, 1.888966],accel_mss,speed_ms,0,blend_radius_m)
    |   movel([0.318366, -1.400186, -2.559168, -0.753034, 1.570796, 1.889162],accel_mss,speed_ms,0,blend_radius_m)
    |   movel([0.318541, -1.400625, -2.558846, -0.752918, 1.570796, 1.889338],accel_mss,speed_ms,0,blend_radius_m)
    |   movel([0.318684, -1.401015, -2.558560, -0.752814, 1.570796, 1.889480],accel_mss,speed_ms,0,blend_radius_m)
    |   movel([0.318813, -1.401414, -2.558266, -0.752708, 1.570796, 1.889610],accel_mss,speed_ms,0,blend_radius_m)
    |   movel([0.318930, -1.401819, -2.557969, -0.752602, 1.570796, 1.889726],accel_mss,speed_ms,0,blend_radius_m)
    |   movel([0.319035, -1.402228, -2.557667, -0.752494, 1.570796, 1.889832],accel_mss,speed_ms,0,blend_radius_m)
    |   movel([0.319122, -1.402613, -2.557383, -0.752392, 1.570796, 1.889918],accel_mss,speed_ms,0,blend_radius_m)
    |   movel([0.319192, -1.403006, -2.557094, -0.752289, 1.570796, 1.889989],accel_mss,speed_ms,0,blend_radius_m)
    |   movel([0.319252, -1.403403, -2.556800, -0.752185, 1.570796, 1.890048],accel_mss,speed_ms,0,blend_radius_m)
    |   movel([0.319295, -1.403808, -2.556501, -0.752080, 1.570796, 1.890091],accel_mss,speed_ms,0,blend_radius_m)
    |   movel([0.319326, -1.404227, -2.556191, -0.751971, 1.570796, 1.890123],accel_mss,speed_ms,0,blend_radius_m)
    |   movel([0.319344, -1.404653, -2.555876, -0.751860, 1.570796, 1.890140],accel_mss,speed_ms,0,blend_radius_m)
    |   movel([0.319347, -1.405081, -2.555559, -0.751749, 1.570796, 1.890143],accel_mss,speed_ms,0,blend_radius_m)
    |   movel([0.319338, -1.405517, -2.555236, -0.751636, 1.570796, 1.890134],accel_mss,speed_ms,0,blend_radius_m)
    |   movel([0.319303, -1.406175, -2.554747, -0.751466, 1.570796, 1.890099],accel_mss,speed_ms,0,blend_radius_m)
    |   movel([0.319250, -1.406838, -2.554255, -0.751296, 1.570796, 1.890046],accel_mss,speed_ms,0,blend_radius_m)
    |   movel([0.319177, -1.407506, -2.553758, -0.751125, 1.570796, 1.889973],accel_mss,speed_ms,0,blend_radius_m)
    |   movel([0.319122, -1.407887, -2.553474, -0.751028, 1.570796, 1.889918],accel_mss,speed_ms,0,blend_radius_m)
    |   movel([0.319055, -1.408269, -2.553190, -0.750931, 1.570796, 1.889852],accel_mss,speed_ms,0,blend_radius_m)
    |   movel([0.318973, -1.408655, -2.552901, -0.750833, 1.570796, 1.889770],accel_mss,speed_ms,0,blend_radius_m)
    |   movel([0.318880, -1.409043, -2.552612, -0.750734, 1.570796, 1.889676],accel_mss,speed_ms,0,blend_radius_m)
    |   movel([0.318769, -1.409433, -2.552320, -0.750636, 1.570796, 1.889566],accel_mss,speed_ms,0,blend_radius_m)
    |   movel([0.318582, -1.410051, -2.551858, -0.750480, 1.570796, 1.889378],accel_mss,speed_ms,0,blend_radius_m)
    |   movel([0.318379, -1.410671, -2.551394, -0.750324, 1.570796, 1.889176],accel_mss,speed_ms,0,blend_radius_m)
    |   movel([0.318164, -1.411292, -2.550929, -0.750169, 1.570796, 1.888960],accel_mss,speed_ms,0,blend_radius_m)
    |   movel([0.317935, -1.411911, -2.550464, -0.750015, 1.570796, 1.888732],accel_mss,speed_ms,0,blend_radius_m)
    |   movel([0.317694, -1.412534, -2.549995, -0.749860, 1.570796, 1.888490],accel_mss,speed_ms,0,blend_radius_m)
    |   movel([0.317439, -1.413158, -2.549526, -0.749705, 1.570796, 1.888236],accel_mss,speed_ms,0,blend_radius_m)
    |   movel([0.317172, -1.413781, -2.549057, -0.749552, 1.570796, 1.887968],accel_mss,speed_ms,0,blend_radius_m)
    |   movel([0.316891, -1.414403, -2.548587, -0.749399, 1.570796, 1.887688],accel_mss,speed_ms,0,blend_radius_m)
    |   movel([0.316702, -1.414803, -2.548285, -0.749301, 1.570796, 1.887499],accel_mss,speed_ms,0,blend_radius_m)
    |   movel([0.316500, -1.415201, -2.547984, -0.749204, 1.570796, 1.887297],accel_mss,speed_ms,0,blend_radius_m)
    |   movel([0.316286, -1.415598, -2.547684, -0.749107, 1.570796, 1.887082],accel_mss,speed_ms,0,blend_radius_m)
    |   movel([0.316060, -1.415994, -2.547385, -0.749011, 1.570796, 1.886857],accel_mss,speed_ms,0,blend_radius_m)
    |   movel([0.315822, -1.416388, -2.547086, -0.748915, 1.570796, 1.886618],accel_mss,speed_ms,0,blend_radius_m)
    |   movel([0.315491, -1.416914, -2.546687, -0.748788, 1.570796, 1.886288],accel_mss,speed_ms,0,blend_radius_m)
    |   movel([0.315149, -1.417434, -2.546292, -0.748662, 1.570796, 1.885946],accel_mss,speed_ms,0,blend_radius_m)
    |   movel([0.314795, -1.417953, -2.545898, -0.748538, 1.570796, 1.885591],accel_mss,speed_ms,0,blend_radius_m)
    |   movel([0.314428, -1.418469, -2.545506, -0.748414, 1.570796, 1.885224],accel_mss,speed_ms,0,blend_radius_m)
    |   movel([0.314052, -1.418980, -2.545116, -0.748292, 1.570796, 1.884848],accel_mss,speed_ms,0,blend_radius_m)
    |   speed_ms = 0.003
    |   movel([0.314052, -1.406365, -2.539347, -0.766677, 1.570796, 1.884848],accel_mss,speed_ms,0,blend_radius_m)
    |   speed_ms = 0.01
    |   movel([0.314052, -1.382109, -2.527415, -0.802865, 1.570796, 1.884848],accel_mss,speed_ms,0,blend_radius_m)
    |   movel([0.312136, -1.381543, -2.527823, -0.803023, 1.570796, 1.882933],accel_mss,speed_ms,0,blend_radius_m)
    |   movel([0.312136, -1.405810, -2.539761, -0.766817, 1.570796, 1.882933],accel_mss,speed_ms,0,blend_radius_m)
    |   speed_ms = 0.003
    |   movel([0.312136, -1.415246, -2.544104, -0.753040, 1.570796, 1.882933],accel_mss,speed_ms,0,blend_radius_m)
    |   speed_ms = 0.007
    |   movel([0.311757, -1.415741, -2.543729, -0.752920, 1.570796, 1.882553],accel_mss,speed_ms,0,blend_radius_m)
    |   movel([0.311364, -1.416228, -2.543359, -0.752802, 1.570796, 1.882161],accel_mss,speed_ms,0,blend_radius_m)
    |   movel([0.310958, -1.416710, -2.542993, -0.752686, 1.570796, 1.881755],accel_mss,speed_ms,0,blend_radius_m)
    |   movel([0.310541, -1.417186, -2.542632, -0.752571, 1.570796, 1.881338],accel_mss,speed_ms,0,blend_radius_m)
    |   movel([0.310112, -1.417655, -2.542275, -0.752459, 1.570796, 1.880908],accel_mss,speed_ms,0,blend_radius_m)
    |   movel([0.309672, -1.418116, -2.541925, -0.752349, 1.570796, 1.880468],accel_mss,speed_ms,0,blend_radius_m)
    |   movel([0.309219, -1.418569, -2.541579, -0.752241, 1.570796, 1.880016],accel_mss,speed_ms,0,blend_radius_m)
    |   movel([0.308758, -1.419015, -2.541239, -0.752135, 1.570796, 1.879555],accel_mss,speed_ms,0,blend_radius_m)
    |   movel([0.308294, -1.419446, -2.540911, -0.752033, 1.570796, 1.879090],accel_mss,speed_ms,0,blend_radius_m)
    |   movel([0.307821, -1.419865, -2.540590, -0.751934, 1.570796, 1.878617],accel_mss,speed_ms,0,blend_radius_m)
    |   movel([0.307339, -1.420277, -2.540276, -0.751837, 1.570796, 1.878136],accel_mss,speed_ms,0,blend_radius_m)
    |   movel([0.306846, -1.420679, -2.539968, -0.751742, 1.570796, 1.877642],accel_mss,speed_ms,0,blend_radius_m)
    |   movel([0.306348, -1.421071, -2.539668, -0.751650, 1.570796, 1.877144],accel_mss,speed_ms,0,blend_radius_m)
    |   movel([0.305840, -1.421451, -2.539377, -0.751561, 1.570796, 1.876637],accel_mss,speed_ms,0,blend_radius_m)
    |   movel([0.305325, -1.421821, -2.539093, -0.751475, 1.570796, 1.876122],accel_mss,speed_ms,0,blend_radius_m)
    |   movel([0.304805, -1.422182, -2.538816, -0.751391, 1.570796, 1.875602],accel_mss,speed_ms,0,blend_radius_m)
    |   movel([0.304285, -1.422524, -2.538554, -0.751311, 1.570796, 1.875081],accel_mss,speed_ms,0,blend_radius_m)
    |   movel([0.303758, -1.422856, -2.538298, -0.751234, 1.570796, 1.874554],accel_mss,speed_ms,0,blend_radius_m)
    |   movel([0.303226, -1.423175, -2.538054, -0.751161, 1.570796, 1.874022],accel_mss,speed_ms,0,blend_radius_m)
    |   movel([0.302690, -1.423481, -2.537818, -0.751090, 1.570796, 1.873487],accel_mss,speed_ms,0,blend_radius_m)
    |   movel([0.302150, -1.423773, -2.537593, -0.751023, 1.570796, 1.872947],accel_mss,speed_ms,0,blend_radius_m)
    |   movel([0.301607, -1.424051, -2.537379, -0.750959, 1.570796, 1.872403],accel_mss,speed_ms,0,blend_radius_m)
    |   movel([0.301058, -1.424318, -2.537174, -0.750897, 1.570796, 1.871855],accel_mss,speed_ms,0,blend_radius_m)
    |   movel([0.300508, -1.424570, -2.536979, -0.750840, 1.570796, 1.871305],accel_mss,speed_ms,0,blend_radius_m)
    |   movel([0.300050, -1.424768, -2.536827, -0.750794, 1.570796, 1.870846],accel_mss,speed_ms,0,blend_radius_m)
    |   movel([0.299593, -1.424953, -2.536684, -0.750752, 1.570796, 1.870390],accel_mss,speed_ms,0,blend_radius_m)
    |   movel([0.299134, -1.425126, -2.536551, -0.750713, 1.570796, 1.869931],accel_mss,speed_ms,0,blend_radius_m)
    |   movel([0.298673, -1.425287, -2.536426, -0.750676, 1.570796, 1.869469],accel_mss,speed_ms,0,blend_radius_m)
    |   movel([0.298216, -1.425435, -2.536312, -0.750642, 1.570796, 1.869012],accel_mss,speed_ms,0,blend_radius_m)
    |   movel([0.297756, -1.425572, -2.536206, -0.750611, 1.570796, 1.868552],accel_mss,speed_ms,0,blend_radius_m)
    |   movel([0.297299, -1.425694, -2.536112, -0.750583, 1.570796, 1.868095],accel_mss,speed_ms,0,blend_radius_m)
    |   movel([0.296735, -1.425832, -2.536005, -0.750552, 1.570796, 1.867531],accel_mss,speed_ms,0,blend_radius_m)
    |   movel([0.296178, -1.425951, -2.535913, -0.750525, 1.570796, 1.866974],accel_mss,speed_ms,0,blend_radius_m)
    |   movel([0.295621, -1.426056, -2.535832, -0.750501, 1.570796, 1.866417],accel_mss,speed_ms,0,blend_radius_m)
    |   movel([0.295067, -1.426145, -2.535763, -0.750481, 1.570796, 1.865863],accel_mss,speed_ms,0,blend_radius_m)
    |   movel([0.294518, -1.426219, -2.535706, -0.750464, 1.570796, 1.865314],accel_mss,speed_ms,0,blend_radius_m)
    |   movel([0.293975, -1.426274, -2.535663, -0.750452, 1.570796, 1.864771],accel_mss,speed_ms,0,blend_radius_m)
    |   movel([0.293435, -1.426316, -2.535631, -0.750442, 1.570796, 1.864231],accel_mss,speed_ms,0,blend_radius_m)
    |   movel([0.292902, -1.426342, -2.535611, -0.750436, 1.570796, 1.863698],accel_mss,speed_ms,0,blend_radius_m)
    |   movel([0.292374, -1.426350, -2.535605, -0.750434, 1.570796, 1.863171],accel_mss,speed_ms,0,blend_radius_m)
    |   movel([0.291854, -1.426343, -2.535610, -0.750436, 1.570796, 1.862650],accel_mss,speed_ms,0,blend_radius_m)
    |   movel([0.291341, -1.426319, -2.535628, -0.750441, 1.570796, 1.862138],accel_mss,speed_ms,0,blend_radius_m)
    |   movel([0.290836, -1.426279, -2.535659, -0.750451, 1.570796, 1.861633],accel_mss,speed_ms,0,blend_radius_m)
    |   movel([0.290434, -1.426233, -2.535695, -0.750461, 1.570796, 1.861231],accel_mss,speed_ms,0,blend_radius_m)
    |   movel([0.290036, -1.426175, -2.535740, -0.750474, 1.570796, 1.860833],accel_mss,speed_ms,0,blend_radius_m)
    |   movel([0.289649, -1.426104, -2.535795, -0.750490, 1.570796, 1.860445],accel_mss,speed_ms,0,blend_radius_m)
    |   movel([0.289269, -1.426017, -2.535862, -0.750510, 1.570796, 1.860065],accel_mss,speed_ms,0,blend_radius_m)
    |   movel([0.288899, -1.425920, -2.535937, -0.750532, 1.570796, 1.859695],accel_mss,speed_ms,0,blend_radius_m)
    |   movel([0.288537, -1.425810, -2.536022, -0.750557, 1.570796, 1.859333],accel_mss,speed_ms,0,blend_radius_m)
    |   movel([0.288184, -1.425685, -2.536119, -0.750585, 1.570796, 1.858980],accel_mss,speed_ms,0,blend_radius_m)
    |   movel([0.287797, -1.425535, -2.536235, -0.750619, 1.570796, 1.858594],accel_mss,speed_ms,0,blend_radius_m)
    |   movel([0.287423, -1.425367, -2.536364, -0.750658, 1.570796, 1.858219],accel_mss,speed_ms,0,blend_radius_m)
    |   movel([0.287057, -1.425190, -2.536501, -0.750698, 1.570796, 1.857854],accel_mss,speed_ms,0,blend_radius_m)
    |   movel([0.286706, -1.424998, -2.536649, -0.750742, 1.570796, 1.857502],accel_mss,speed_ms,0,blend_radius_m)
    |   movel([0.286365, -1.424793, -2.536807, -0.750789, 1.570796, 1.857161],accel_mss,speed_ms,0,blend_radius_m)
    |   movel([0.286034, -1.424576, -2.536974, -0.750838, 1.570796, 1.856830],accel_mss,speed_ms,0,blend_radius_m)
    |   movel([0.285718, -1.424346, -2.537152, -0.750891, 1.570796, 1.856514],accel_mss,speed_ms,0,blend_radius_m)
    |   movel([0.285414, -1.424105, -2.537338, -0.750946, 1.570796, 1.856210],accel_mss,speed_ms,0,blend_radius_m)
    |   movel([0.285121, -1.423852, -2.537532, -0.751004, 1.570796, 1.855917],accel_mss,speed_ms,0,blend_radius_m)
    |   movel([0.284844, -1.423588, -2.537736, -0.751065, 1.570796, 1.855640],accel_mss,speed_ms,0,blend_radius_m)
    |   movel([0.284578, -1.423310, -2.537950, -0.751129, 1.570796, 1.855374],accel_mss,speed_ms,0,blend_radius_m)
    |   movel([0.284328, -1.423022, -2.538171, -0.751196, 1.570796, 1.855124],accel_mss,speed_ms,0,blend_radius_m)
    |   movel([0.284060, -1.422685, -2.538430, -0.751274, 1.570796, 1.854856],accel_mss,speed_ms,0,blend_radius_m)
    |   movel([0.283809, -1.422336, -2.538698, -0.751355, 1.570796, 1.854606],accel_mss,speed_ms,0,blend_radius_m)
    |   movel([0.283573, -1.421975, -2.538975, -0.751439, 1.570796, 1.854369],accel_mss,speed_ms,0,blend_radius_m)
    |   movel([0.283355, -1.421604, -2.539259, -0.751525, 1.570796, 1.854151],accel_mss,speed_ms,0,blend_radius_m)
    |   movel([0.283152, -1.421222, -2.539553, -0.751615, 1.570796, 1.853948],accel_mss,speed_ms,0,blend_radius_m)
    |   movel([0.282965, -1.420827, -2.539855, -0.751707, 1.570796, 1.853762],accel_mss,speed_ms,0,blend_radius_m)
    |   movel([0.282798, -1.420421, -2.540165, -0.751803, 1.570796, 1.853594],accel_mss,speed_ms,0,blend_radius_m)
    |   movel([0.282645, -1.420008, -2.540481, -0.751900, 1.570796, 1.853442],accel_mss,speed_ms,0,blend_radius_m)
    |   movel([0.282512, -1.419583, -2.540806, -0.752000, 1.570796, 1.853309],accel_mss,speed_ms,0,blend_radius_m)
    |   movel([0.282395, -1.419149, -2.541137, -0.752103, 1.570796, 1.853191],accel_mss,speed_ms,0,blend_radius_m)
    |   movel([0.282296, -1.418707, -2.541474, -0.752208, 1.570796, 1.853092],accel_mss,speed_ms,0,blend_radius_m)
    |   movel([0.282212, -1.418249, -2.541823, -0.752317, 1.570796, 1.853009],accel_mss,speed_ms,0,blend_radius_m)
    |   movel([0.282147, -1.417782, -2.542178, -0.752428, 1.570796, 1.852944],accel_mss,speed_ms,0,blend_radius_m)
    |   movel([0.282100, -1.417308, -2.542539, -0.752542, 1.570796, 1.852896],accel_mss,speed_ms,0,blend_radius_m)
    |   movel([0.282070, -1.416826, -2.542905, -0.752658, 1.570796, 1.852867],accel_mss,speed_ms,0,blend_radius_m)
    |   movel([0.282060, -1.416339, -2.543275, -0.752775, 1.570796, 1.852857],accel_mss,speed_ms,0,blend_radius_m)
    |   movel([0.282066, -1.415843, -2.543651, -0.752895, 1.570796, 1.852863],accel_mss,speed_ms,0,blend_radius_m)
    |   movel([0.282091, -1.415343, -2.544030, -0.753016, 1.570796, 1.852888],accel_mss,speed_ms,0,blend_radius_m)
    |   movel([0.282135, -1.414834, -2.544415, -0.753140, 1.570796, 1.852931],accel_mss,speed_ms,0,blend_radius_m)
    |   movel([0.282194, -1.414323, -2.544802, -0.753265, 1.570796, 1.852990],accel_mss,speed_ms,0,blend_radius_m)
    |   movel([0.282274, -1.413805, -2.545193, -0.753391, 1.570796, 1.853070],accel_mss,speed_ms,0,blend_radius_m)
    |   movel([0.282370, -1.413283, -2.545586, -0.753519, 1.570796, 1.853166],accel_mss,speed_ms,0,blend_radius_m)
    |   movel([0.282484, -1.412761, -2.545980, -0.753648, 1.570796, 1.853281],accel_mss,speed_ms,0,blend_radius_m)
    |   movel([0.282618, -1.412237, -2.546375, -0.753777, 1.570796, 1.853414],accel_mss,speed_ms,0,blend_radius_m)
    |   movel([0.282767, -1.411710, -2.546771, -0.753908, 1.570796, 1.853563],accel_mss,speed_ms,0,blend_radius_m)
    |   movel([0.282934, -1.411179, -2.547170, -0.754040, 1.570796, 1.853730],accel_mss,speed_ms,0,blend_radius_m)
    |   movel([0.283121, -1.410648, -2.547569, -0.754172, 1.570796, 1.853917],accel_mss,speed_ms,0,blend_radius_m)
    |   movel([0.283324, -1.410114, -2.547969, -0.754306, 1.570796, 1.854121],accel_mss,speed_ms,0,blend_radius_m)
    |   movel([0.283547, -1.409578, -2.548371, -0.754440, 1.570796, 1.854343],accel_mss,speed_ms,0,blend_radius_m)
    |   movel([0.283785, -1.409041, -2.548772, -0.754575, 1.570796, 1.854581],accel_mss,speed_ms,0,blend_radius_m)
    |   movel([0.284041, -1.408507, -2.549172, -0.754710, 1.570796, 1.854837],accel_mss,speed_ms,0,blend_radius_m)
    |   movel([0.284312, -1.407973, -2.549571, -0.754846, 1.570796, 1.855109],accel_mss,speed_ms,0,blend_radius_m)
    |   movel([0.284603, -1.407438, -2.549969, -0.754982, 1.570796, 1.855399],accel_mss,speed_ms,0,blend_radius_m)
    |   movel([0.284890, -1.406932, -2.550346, -0.755110, 1.570796, 1.855687],accel_mss,speed_ms,0,blend_radius_m)
    |   movel([0.285189, -1.406427, -2.550722, -0.755239, 1.570796, 1.855986],accel_mss,speed_ms,0,blend_radius_m)
    |   movel([0.285499, -1.405925, -2.551096, -0.755368, 1.570796, 1.856296],accel_mss,speed_ms,0,blend_radius_m)
    |   movel([0.285820, -1.405425, -2.551467, -0.755497, 1.570796, 1.856616],accel_mss,speed_ms,0,blend_radius_m)
    |   movel([0.286154, -1.404926, -2.551838, -0.755625, 1.570796, 1.856950],accel_mss,speed_ms,0,blend_radius_m)
    |   movel([0.286465, -1.404479, -2.552169, -0.755741, 1.570796, 1.857261],accel_mss,speed_ms,0,blend_radius_m)
    |   movel([0.286788, -1.404035, -2.552498, -0.755856, 1.570796, 1.857585],accel_mss,speed_ms,0,blend_radius_m)
    |   movel([0.287125, -1.403595, -2.552823, -0.755970, 1.570796, 1.857921],accel_mss,speed_ms,0,blend_radius_m)
    |   movel([0.287473, -1.403160, -2.553145, -0.756083, 1.570796, 1.858269],accel_mss,speed_ms,0,blend_radius_m)
    |   movel([0.287831, -1.402731, -2.553463, -0.756196, 1.570796, 1.858628],accel_mss,speed_ms,0,blend_radius_m)
    |   movel([0.288198, -1.402310, -2.553773, -0.756306, 1.570796, 1.858994],accel_mss,speed_ms,0,blend_radius_m)
    |   movel([0.288577, -1.401897, -2.554078, -0.756414, 1.570796, 1.859373],accel_mss,speed_ms,0,blend_radius_m)
    |   movel([0.288965, -1.401488, -2.554379, -0.756522, 1.570796, 1.859761],accel_mss,speed_ms,0,blend_radius_m)
    |   movel([0.289365, -1.401087, -2.554675, -0.756627, 1.570796, 1.860161],accel_mss,speed_ms,0,blend_radius_m)
    |   movel([0.289772, -1.400693, -2.554964, -0.756731, 1.570796, 1.860568],accel_mss,speed_ms,0,blend_radius_m)
    |   movel([0.290226, -1.400273, -2.555273, -0.756842, 1.570796, 1.861023],accel_mss,speed_ms,0,blend_radius_m)
    |   movel([0.290686, -1.399859, -2.555578, -0.756952, 1.570796, 1.861482],accel_mss,speed_ms,0,blend_radius_m)
    |   movel([0.291155, -1.399452, -2.555877, -0.757061, 1.570796, 1.861951],accel_mss,speed_ms,0,blend_radius_m)
    |   movel([0.291630, -1.399052, -2.556170, -0.757167, 1.570796, 1.862427],accel_mss,speed_ms,0,blend_radius_m)
    |   movel([0.292111, -1.398661, -2.556457, -0.757272, 1.570796, 1.862907],accel_mss,speed_ms,0,blend_radius_m)
    |   movel([0.292598, -1.398277, -2.556738, -0.757375, 1.570796, 1.863394],accel_mss,speed_ms,0,blend_radius_m)
    |   movel([0.293092, -1.397900, -2.557013, -0.757475, 1.570796, 1.863888],accel_mss,speed_ms,0,blend_radius_m)
    |   movel([0.293591, -1.397532, -2.557283, -0.757574, 1.570796, 1.864387],accel_mss,speed_ms,0,blend_radius_m)
    |   movel([0.294094, -1.397171, -2.557546, -0.757671, 1.570796, 1.864890],accel_mss,speed_ms,0,blend_radius_m)
    |   movel([0.294554, -1.396854, -2.557778, -0.757757, 1.570796, 1.865351],accel_mss,speed_ms,0,blend_radius_m)
    |   movel([0.295017, -1.396548, -2.558001, -0.757840, 1.570796, 1.865814],accel_mss,speed_ms,0,blend_radius_m)
    |   movel([0.295488, -1.396255, -2.558215, -0.757919, 1.570796, 1.866285],accel_mss,speed_ms,0,blend_radius_m)
    |   movel([0.295964, -1.395970, -2.558423, -0.757996, 1.570796, 1.866760],accel_mss,speed_ms,0,blend_radius_m)
    |   movel([0.296434, -1.395702, -2.558618, -0.758069, 1.570796, 1.867230],accel_mss,speed_ms,0,blend_radius_m)
    |   movel([0.296912, -1.395444, -2.558805, -0.758139, 1.570796, 1.867708],accel_mss,speed_ms,0,blend_radius_m)
    |   movel([0.297390, -1.395199, -2.558984, -0.758206, 1.570796, 1.868187],accel_mss,speed_ms,0,blend_radius_m)
    |   movel([0.297872, -1.394967, -2.559153, -0.758269, 1.570796, 1.868669],accel_mss,speed_ms,0,blend_radius_m)
    |   movel([0.298398, -1.394726, -2.559328, -0.758335, 1.570796, 1.869194],accel_mss,speed_ms,0,blend_radius_m)
    |   movel([0.298923, -1.394496, -2.559495, -0.758398, 1.570796, 1.869719],accel_mss,speed_ms,0,blend_radius_m)
    |   movel([0.299450, -1.394278, -2.559653, -0.758457, 1.570796, 1.870246],accel_mss,speed_ms,0,blend_radius_m)
    |   movel([0.299980, -1.394069, -2.559805, -0.758515, 1.570796, 1.870776],accel_mss,speed_ms,0,blend_radius_m)
    |   movel([0.300614, -1.393833, -2.559977, -0.758579, 1.570796, 1.871411],accel_mss,speed_ms,0,blend_radius_m)
    |   movel([0.301249, -1.393612, -2.560137, -0.758640, 1.570796, 1.872045],accel_mss,speed_ms,0,blend_radius_m)
    |   movel([0.301536, -1.393521, -2.560203, -0.758665, 1.570796, 1.872333],accel_mss,speed_ms,0,blend_radius_m)
    |   movel([0.301823, -1.393441, -2.560261, -0.758687, 1.570796, 1.872619],accel_mss,speed_ms,0,blend_radius_m)
    |   movel([0.302107, -1.393375, -2.560309, -0.758705, 1.570796, 1.872904],accel_mss,speed_ms,0,blend_radius_m)
    |   movel([0.302431, -1.393313, -2.560354, -0.758722, 1.570796, 1.873228],accel_mss,speed_ms,0,blend_radius_m)
    |   movel([0.302757, -1.393260, -2.560392, -0.758737, 1.570796, 1.873553],accel_mss,speed_ms,0,blend_radius_m)
    |   movel([0.303077, -1.393218, -2.560423, -0.758748, 1.570796, 1.873873],accel_mss,speed_ms,0,blend_radius_m)
    |   movel([0.304031, -1.393115, -2.560497, -0.758777, 1.570796, 1.874827],accel_mss,speed_ms,0,blend_radius_m)
    |   movel([0.304981, -1.393021, -2.560565, -0.758803, 1.570796, 1.875778],accel_mss,speed_ms,0,blend_radius_m)
    |   movel([0.305935, -1.392932, -2.560629, -0.758827, 1.570796, 1.876732],accel_mss,speed_ms,0,blend_radius_m)
    |   movel([0.306883, -1.392856, -2.560685, -0.758848, 1.570796, 1.877679],accel_mss,speed_ms,0,blend_radius_m)
    |   movel([0.307197, -1.392837, -2.560698, -0.758853, 1.570796, 1.877994],accel_mss,speed_ms,0,blend_radius_m)
    |   movel([0.307506, -1.392827, -2.560705, -0.758856, 1.570796, 1.878303],accel_mss,speed_ms,0,blend_radius_m)
    |   movel([0.307811, -1.392831, -2.560703, -0.758855, 1.570796, 1.878607],accel_mss,speed_ms,0,blend_radius_m)
    |   movel([0.308070, -1.392848, -2.560691, -0.758850, 1.570796, 1.878866],accel_mss,speed_ms,0,blend_radius_m)
    |   movel([0.308323, -1.392876, -2.560670, -0.758843, 1.570796, 1.879119],accel_mss,speed_ms,0,blend_radius_m)
    |   movel([0.308569, -1.392918, -2.560640, -0.758831, 1.570796, 1.879365],accel_mss,speed_ms,0,blend_radius_m)
    |   movel([0.309105, -1.393031, -2.560558, -0.758800, 1.570796, 1.879901],accel_mss,speed_ms,0,blend_radius_m)
    |   movel([0.309633, -1.393161, -2.560464, -0.758764, 1.570796, 1.880430],accel_mss,speed_ms,0,blend_radius_m)
    |   movel([0.310064, -1.393283, -2.560375, -0.758731, 1.570796, 1.880860],accel_mss,speed_ms,0,blend_radius_m)
    |   movel([0.310487, -1.393419, -2.560277, -0.758693, 1.570796, 1.881284],accel_mss,speed_ms,0,blend_radius_m)
    |   movel([0.310896, -1.393571, -2.560167, -0.758651, 1.570796, 1.881692],accel_mss,speed_ms,0,blend_radius_m)
    |   movel([0.311296, -1.393735, -2.560048, -0.758606, 1.570796, 1.882092],accel_mss,speed_ms,0,blend_radius_m)
    |   movel([0.311683, -1.393915, -2.559917, -0.758557, 1.570796, 1.882480],accel_mss,speed_ms,0,blend_radius_m)
    |   movel([0.312059, -1.394107, -2.559778, -0.758504, 1.570796, 1.882856],accel_mss,speed_ms,0,blend_radius_m)
    |   movel([0.312421, -1.394315, -2.559627, -0.758447, 1.570796, 1.883217],accel_mss,speed_ms,0,blend_radius_m)
    |   movel([0.312771, -1.394535, -2.559467, -0.758387, 1.570796, 1.883567],accel_mss,speed_ms,0,blend_radius_m)
    |   movel([0.313107, -1.394770, -2.559296, -0.758323, 1.570796, 1.883903],accel_mss,speed_ms,0,blend_radius_m)
    |   movel([0.313432, -1.395016, -2.559117, -0.758256, 1.570796, 1.884228],accel_mss,speed_ms,0,blend_radius_m)
    |   movel([0.313741, -1.395277, -2.558928, -0.758185, 1.570796, 1.884537],accel_mss,speed_ms,0,blend_radius_m)
    |   movel([0.314036, -1.395549, -2.558729, -0.758111, 1.570796, 1.884832],accel_mss,speed_ms,0,blend_radius_m)
    |   movel([0.314348, -1.395863, -2.558501, -0.758025, 1.570796, 1.885144],accel_mss,speed_ms,0,blend_radius_m)
    |   movel([0.314641, -1.396194, -2.558260, -0.757936, 1.570796, 1.885437],accel_mss,speed_ms,0,blend_radius_m)
    |   movel([0.314920, -1.396536, -2.558010, -0.757843, 1.570796, 1.885716],accel_mss,speed_ms,0,blend_radius_m)
    |   movel([0.315178, -1.396893, -2.557749, -0.757747, 1.570796, 1.885974],accel_mss,speed_ms,0,blend_radius_m)
    |   movel([0.315421, -1.397260, -2.557481, -0.757648, 1.570796, 1.886217],accel_mss,speed_ms,0,blend_radius_m)
    |   movel([0.315645, -1.397641, -2.557203, -0.757545, 1.570796, 1.886442],accel_mss,speed_ms,0,blend_radius_m)
    |   movel([0.315851, -1.398035, -2.556915, -0.757439, 1.570796, 1.886648],accel_mss,speed_ms,0,blend_radius_m)
    |   movel([0.316037, -1.398440, -2.556618, -0.757331, 1.570796, 1.886834],accel_mss,speed_ms,0,blend_radius_m)
    |   movel([0.316208, -1.398855, -2.556314, -0.757220, 1.570796, 1.887005],accel_mss,speed_ms,0,blend_radius_m)
    |   movel([0.316357, -1.399281, -2.556002, -0.757106, 1.570796, 1.887154],accel_mss,speed_ms,0,blend_radius_m)
    |   movel([0.316491, -1.399718, -2.555681, -0.756990, 1.570796, 1.887287],accel_mss,speed_ms,0,blend_radius_m)
    |   movel([0.316605, -1.400171, -2.555348, -0.756870, 1.570796, 1.887401],accel_mss,speed_ms,0,blend_radius_m)
    |   movel([0.316701, -1.400634, -2.555008, -0.756747, 1.570796, 1.887498],accel_mss,speed_ms,0,blend_radius_m)
    |   movel([0.316779, -1.401105, -2.554661, -0.756623, 1.570796, 1.887576],accel_mss,speed_ms,0,blend_radius_m)
    |   movel([0.316839, -1.401584, -2.554309, -0.756497, 1.570796, 1.887635],accel_mss,speed_ms,0,blend_radius_m)
    |   movel([0.316877, -1.402072, -2.553949, -0.756368, 1.570796, 1.887673],accel_mss,speed_ms,0,blend_radius_m)
    |   movel([0.316899, -1.402565, -2.553585, -0.756239, 1.570796, 1.887695],accel_mss,speed_ms,0,blend_radius_m)
    |   movel([0.316900, -1.403067, -2.553214, -0.756108, 1.570796, 1.887697],accel_mss,speed_ms,0,blend_radius_m)
    |   movel([0.316884, -1.403573, -2.552840, -0.755976, 1.570796, 1.887680],accel_mss,speed_ms,0,blend_radius_m)
    |   movel([0.316848, -1.404085, -2.552461, -0.755843, 1.570796, 1.887644],accel_mss,speed_ms,0,blend_radius_m)
    |   movel([0.316794, -1.404603, -2.552077, -0.755709, 1.570796, 1.887590],accel_mss,speed_ms,0,blend_radius_m)
    |   movel([0.316720, -1.405125, -2.551690, -0.755574, 1.570796, 1.887516],accel_mss,speed_ms,0,blend_radius_m)
    |   movel([0.316626, -1.405658, -2.551294, -0.755437, 1.570796, 1.887423],accel_mss,speed_ms,0,blend_radius_m)
    |   movel([0.316516, -1.406193, -2.550896, -0.755299, 1.570796, 1.887313],accel_mss,speed_ms,0,blend_radius_m)
    |   movel([0.316386, -1.406734, -2.550494, -0.755161, 1.570796, 1.887183],accel_mss,speed_ms,0,blend_radius_m)
    |   movel([0.316241, -1.407273, -2.550092, -0.755023, 1.570796, 1.887038],accel_mss,speed_ms,0,blend_radius_m)
    |   movel([0.316077, -1.407818, -2.549686, -0.754885, 1.570796, 1.886873],accel_mss,speed_ms,0,blend_radius_m)
    |   movel([0.315894, -1.408362, -2.549280, -0.754747, 1.570796, 1.886690],accel_mss,speed_ms,0,blend_radius_m)
    |   movel([0.315695, -1.408908, -2.548872, -0.754609, 1.570796, 1.886491],accel_mss,speed_ms,0,blend_radius_m)
    |   movel([0.315481, -1.409453, -2.548464, -0.754472, 1.570796, 1.886277],accel_mss,speed_ms,0,blend_radius_m)
    |   movel([0.315246, -1.410000, -2.548055, -0.754334, 1.570796, 1.886043],accel_mss,speed_ms,0,blend_radius_m)
    |   movel([0.314999, -1.410545, -2.547646, -0.754198, 1.570796, 1.885795],accel_mss,speed_ms,0,blend_radius_m)
    |   movel([0.314734, -1.411088, -2.547238, -0.754062, 1.570796, 1.885531],accel_mss,speed_ms,0,blend_radius_m)
    |   movel([0.314459, -1.411618, -2.546840, -0.753931, 1.570796, 1.885255],accel_mss,speed_ms,0,blend_radius_m)
    |   movel([0.314169, -1.412146, -2.546443, -0.753800, 1.570796, 1.884965],accel_mss,speed_ms,0,blend_radius_m)
    |   movel([0.313867, -1.412670, -2.546048, -0.753670, 1.570796, 1.884663],accel_mss,speed_ms,0,blend_radius_m)
    |   movel([0.313547, -1.413194, -2.545654, -0.753541, 1.570796, 1.884343],accel_mss,speed_ms,0,blend_radius_m)
    |   movel([0.313216, -1.413713, -2.545262, -0.753414, 1.570796, 1.884012],accel_mss,speed_ms,0,blend_radius_m)
    |   movel([0.312869, -1.414228, -2.544873, -0.753288, 1.570796, 1.883665],accel_mss,speed_ms,0,blend_radius_m)
    |   movel([0.312509, -1.414740, -2.544486, -0.753163, 1.570796, 1.883305],accel_mss,speed_ms,0,blend_radius_m)
    |   movel([0.312136, -1.415246, -2.544104, -0.753040, 1.570796, 1.882933],accel_mss,speed_ms,0,blend_radius_m)
    |   speed_ms = 0.003
    |   movel([0.312136, -1.418431, -2.545534, -0.748423, 1.570796, 1.882933],accel_mss,speed_ms,0,blend_radius_m)
    |   speed_ms = 0.007
    |   movel([0.311757, -1.418925, -2.545158, -0.748305, 1.570796, 1.882553],accel_mss,speed_ms,0,blend_radius_m)
    |   movel([0.311364, -1.419411, -2.544788, -0.748190, 1.570796, 1.882161],accel_mss,speed_ms,0,blend_radius_m)
    |   movel([0.310958, -1.419892, -2.544422, -0.748076, 1.570796, 1.881755],accel_mss,speed_ms,0,blend_radius_m)
    |   movel([0.310541, -1.420366, -2.544059, -0.747963, 1.570796, 1.881338],accel_mss,speed_ms,0,blend_radius_m)
    |   movel([0.310112, -1.420834, -2.543702, -0.747853, 1.570796, 1.880908],accel_mss,speed_ms,0,blend_radius_m)
    |   movel([0.309672, -1.421293, -2.543351, -0.747745, 1.570796, 1.880468],accel_mss,speed_ms,0,blend_radius_m)
    |   movel([0.309219, -1.421745, -2.543005, -0.747639, 1.570796, 1.880016],accel_mss,speed_ms,0,blend_radius_m)
    |   movel([0.308758, -1.422190, -2.542664, -0.747535, 1.570796, 1.879555],accel_mss,speed_ms,0,blend_radius_m)
    |   movel([0.308294, -1.422620, -2.542334, -0.747435, 1.570796, 1.879090],accel_mss,speed_ms,0,blend_radius_m)
    |   movel([0.307821, -1.423038, -2.542014, -0.747338, 1.570796, 1.878617],accel_mss,speed_ms,0,blend_radius_m)
    |   movel([0.307339, -1.423448, -2.541698, -0.747242, 1.570796, 1.878136],accel_mss,speed_ms,0,blend_radius_m)
    |   movel([0.306846, -1.423849, -2.541390, -0.747150, 1.570796, 1.877642],accel_mss,speed_ms,0,blend_radius_m)
    |   movel([0.306348, -1.424240, -2.541090, -0.747059, 1.570796, 1.877144],accel_mss,speed_ms,0,blend_radius_m)
    |   movel([0.305840, -1.424619, -2.540798, -0.746972, 1.570796, 1.876637],accel_mss,speed_ms,0,blend_radius_m)
    |   movel([0.305325, -1.424989, -2.540513, -0.746887, 1.570796, 1.876122],accel_mss,speed_ms,0,blend_radius_m)
    |   movel([0.304805, -1.425348, -2.540236, -0.746805, 1.570796, 1.875602],accel_mss,speed_ms,0,blend_radius_m)
    |   movel([0.304285, -1.425689, -2.539973, -0.746727, 1.570796, 1.875081],accel_mss,speed_ms,0,blend_radius_m)
    |   movel([0.303758, -1.426020, -2.539717, -0.746652, 1.570796, 1.874554],accel_mss,speed_ms,0,blend_radius_m)
    |   movel([0.303226, -1.426338, -2.539472, -0.746579, 1.570796, 1.874022],accel_mss,speed_ms,0,blend_radius_m)
    |   movel([0.302690, -1.426643, -2.539236, -0.746510, 1.570796, 1.873487],accel_mss,speed_ms,0,blend_radius_m)
    |   movel([0.302150, -1.426935, -2.539010, -0.746444, 1.570796, 1.872947],accel_mss,speed_ms,0,blend_radius_m)
    |   movel([0.301607, -1.427212, -2.538796, -0.746381, 1.570796, 1.872403],accel_mss,speed_ms,0,blend_radius_m)
    |   movel([0.301058, -1.427478, -2.538590, -0.746321, 1.570796, 1.871855],accel_mss,speed_ms,0,blend_radius_m)
    |   movel([0.300508, -1.427729, -2.538395, -0.746265, 1.570796, 1.871305],accel_mss,speed_ms,0,blend_radius_m)
    |   movel([0.300050, -1.427926, -2.538242, -0.746220, 1.570796, 1.870846],accel_mss,speed_ms,0,blend_radius_m)
    |   movel([0.299593, -1.428111, -2.538099, -0.746179, 1.570796, 1.870390],accel_mss,speed_ms,0,blend_radius_m)
    |   movel([0.299134, -1.428283, -2.537966, -0.746140, 1.570796, 1.869931],accel_mss,speed_ms,0,blend_radius_m)
    |   movel([0.298673, -1.428444, -2.537841, -0.746104, 1.570796, 1.869469],accel_mss,speed_ms,0,blend_radius_m)
    |   movel([0.298216, -1.428592, -2.537726, -0.746071, 1.570796, 1.869012],accel_mss,speed_ms,0,blend_radius_m)
    |   movel([0.297756, -1.428728, -2.537620, -0.746040, 1.570796, 1.868552],accel_mss,speed_ms,0,blend_radius_m)
    |   movel([0.297299, -1.428850, -2.537526, -0.746013, 1.570796, 1.868095],accel_mss,speed_ms,0,blend_radius_m)
    |   movel([0.296735, -1.428988, -2.537419, -0.745982, 1.570796, 1.867531],accel_mss,speed_ms,0,blend_radius_m)
    |   movel([0.296178, -1.429106, -2.537327, -0.745956, 1.570796, 1.866974],accel_mss,speed_ms,0,blend_radius_m)
    |   movel([0.295621, -1.429211, -2.537245, -0.745933, 1.570796, 1.866417],accel_mss,speed_ms,0,blend_radius_m)
    |   movel([0.295067, -1.429299, -2.537177, -0.745913, 1.570796, 1.865863],accel_mss,speed_ms,0,blend_radius_m)
    |   movel([0.294518, -1.429373, -2.537119, -0.745896, 1.570796, 1.865314],accel_mss,speed_ms,0,blend_radius_m)
    |   movel([0.293975, -1.429429, -2.537076, -0.745884, 1.570796, 1.864771],accel_mss,speed_ms,0,blend_radius_m)
    |   movel([0.293435, -1.429470, -2.537044, -0.745875, 1.570796, 1.864231],accel_mss,speed_ms,0,blend_radius_m)
    |   movel([0.292902, -1.429496, -2.537024, -0.745869, 1.570796, 1.863698],accel_mss,speed_ms,0,blend_radius_m)
    |   movel([0.292374, -1.429504, -2.537018, -0.745867, 1.570796, 1.863171],accel_mss,speed_ms,0,blend_radius_m)
    |   movel([0.291854, -1.429497, -2.537023, -0.745869, 1.570796, 1.862650],accel_mss,speed_ms,0,blend_radius_m)
    |   movel([0.291341, -1.429474, -2.537041, -0.745874, 1.570796, 1.862138],accel_mss,speed_ms,0,blend_radius_m)
    |   movel([0.290836, -1.429433, -2.537073, -0.745883, 1.570796, 1.861633],accel_mss,speed_ms,0,blend_radius_m)
    |   movel([0.290434, -1.429388, -2.537108, -0.745893, 1.570796, 1.861231],accel_mss,speed_ms,0,blend_radius_m)
    |   movel([0.290036, -1.429330, -2.537153, -0.745906, 1.570796, 1.860833],accel_mss,speed_ms,0,blend_radius_m)
    |   movel([0.289649, -1.429258, -2.537209, -0.745922, 1.570796, 1.860445],accel_mss,speed_ms,0,blend_radius_m)
    |   movel([0.289269, -1.429172, -2.537275, -0.745941, 1.570796, 1.860065],accel_mss,speed_ms,0,blend_radius_m)
    |   movel([0.288899, -1.429076, -2.537351, -0.745963, 1.570796, 1.859695],accel_mss,speed_ms,0,blend_radius_m)
    |   movel([0.288537, -1.428966, -2.537436, -0.745987, 1.570796, 1.859333],accel_mss,speed_ms,0,blend_radius_m)
    |   movel([0.288184, -1.428841, -2.537533, -0.746015, 1.570796, 1.858980],accel_mss,speed_ms,0,blend_radius_m)
    |   movel([0.287797, -1.428691, -2.537649, -0.746049, 1.570796, 1.858594],accel_mss,speed_ms,0,blend_radius_m)
    |   movel([0.287423, -1.428524, -2.537779, -0.746086, 1.570796, 1.858219],accel_mss,speed_ms,0,blend_radius_m)
    |   movel([0.287057, -1.428348, -2.537916, -0.746126, 1.570796, 1.857854],accel_mss,speed_ms,0,blend_radius_m)
    |   movel([0.286706, -1.428156, -2.538064, -0.746169, 1.570796, 1.857502],accel_mss,speed_ms,0,blend_radius_m)
    |   movel([0.286365, -1.427951, -2.538223, -0.746215, 1.570796, 1.857161],accel_mss,speed_ms,0,blend_radius_m)
    |   movel([0.286034, -1.427736, -2.538390, -0.746263, 1.570796, 1.856830],accel_mss,speed_ms,0,blend_radius_m)
    |   movel([0.285718, -1.427506, -2.538568, -0.746315, 1.570796, 1.856514],accel_mss,speed_ms,0,blend_radius_m)
    |   movel([0.285414, -1.427265, -2.538754, -0.746369, 1.570796, 1.856210],accel_mss,speed_ms,0,blend_radius_m)
    |   movel([0.285121, -1.427014, -2.538949, -0.746426, 1.570796, 1.855917],accel_mss,speed_ms,0,blend_radius_m)
    |   movel([0.284844, -1.426750, -2.539153, -0.746486, 1.570796, 1.855640],accel_mss,speed_ms,0,blend_radius_m)
    |   movel([0.284578, -1.426473, -2.539368, -0.746549, 1.570796, 1.855374],accel_mss,speed_ms,0,blend_radius_m)
    |   movel([0.284328, -1.426186, -2.539589, -0.746614, 1.570796, 1.855124],accel_mss,speed_ms,0,blend_radius_m)
    |   movel([0.284060, -1.425850, -2.539849, -0.746690, 1.570796, 1.854856],accel_mss,speed_ms,0,blend_radius_m)
    |   movel([0.283809, -1.425502, -2.540117, -0.746770, 1.570796, 1.854606],accel_mss,speed_ms,0,blend_radius_m)
    |   movel([0.283573, -1.425142, -2.540395, -0.746852, 1.570796, 1.854369],accel_mss,speed_ms,0,blend_radius_m)
    |   movel([0.283355, -1.424772, -2.540680, -0.746937, 1.570796, 1.854151],accel_mss,speed_ms,0,blend_radius_m)
    |   movel([0.283152, -1.424390, -2.540974, -0.747025, 1.570796, 1.853948],accel_mss,speed_ms,0,blend_radius_m)
    |   movel([0.282965, -1.423997, -2.541277, -0.747116, 1.570796, 1.853762],accel_mss,speed_ms,0,blend_radius_m)
    |   movel([0.282798, -1.423593, -2.541587, -0.747209, 1.570796, 1.853594],accel_mss,speed_ms,0,blend_radius_m)
    |   movel([0.282645, -1.423181, -2.541904, -0.747304, 1.570796, 1.853442],accel_mss,speed_ms,0,blend_radius_m)
    |   movel([0.282512, -1.422756, -2.542230, -0.747403, 1.570796, 1.853309],accel_mss,speed_ms,0,blend_radius_m)
    |   movel([0.282395, -1.422324, -2.542561, -0.747504, 1.570796, 1.853191],accel_mss,speed_ms,0,blend_radius_m)
    |   movel([0.282296, -1.421883, -2.542899, -0.747607, 1.570796, 1.853092],accel_mss,speed_ms,0,blend_radius_m)
    |   movel([0.282212, -1.421426, -2.543249, -0.747714, 1.570796, 1.853009],accel_mss,speed_ms,0,blend_radius_m)
    |   movel([0.282147, -1.420961, -2.543605, -0.747823, 1.570796, 1.852944],accel_mss,speed_ms,0,blend_radius_m)
    |   movel([0.282100, -1.420488, -2.543967, -0.747935, 1.570796, 1.852896],accel_mss,speed_ms,0,blend_radius_m)
    |   movel([0.282070, -1.420008, -2.544333, -0.748048, 1.570796, 1.852867],accel_mss,speed_ms,0,blend_radius_m)
    |   movel([0.282060, -1.419522, -2.544704, -0.748164, 1.570796, 1.852857],accel_mss,speed_ms,0,blend_radius_m)
    |   movel([0.282066, -1.419027, -2.545081, -0.748281, 1.570796, 1.852863],accel_mss,speed_ms,0,blend_radius_m)
    |   movel([0.282091, -1.418528, -2.545461, -0.748400, 1.570796, 1.852888],accel_mss,speed_ms,0,blend_radius_m)
    |   movel([0.282135, -1.418021, -2.545847, -0.748522, 1.570796, 1.852931],accel_mss,speed_ms,0,blend_radius_m)
    |   movel([0.282194, -1.417511, -2.546234, -0.748644, 1.570796, 1.852990],accel_mss,speed_ms,0,blend_radius_m)
    |   movel([0.282274, -1.416995, -2.546625, -0.748768, 1.570796, 1.853070],accel_mss,speed_ms,0,blend_radius_m)
    |   movel([0.282370, -1.416475, -2.547020, -0.748894, 1.570796, 1.853166],accel_mss,speed_ms,0,blend_radius_m)
    |   movel([0.282484, -1.415954, -2.547414, -0.749020, 1.570796, 1.853281],accel_mss,speed_ms,0,blend_radius_m)
    |   movel([0.282618, -1.415431, -2.547810, -0.749148, 1.570796, 1.853414],accel_mss,speed_ms,0,blend_radius_m)
    |   movel([0.282767, -1.414906, -2.548207, -0.749276, 1.570796, 1.853563],accel_mss,speed_ms,0,blend_radius_m)
    |   movel([0.282934, -1.414376, -2.548607, -0.749405, 1.570796, 1.853730],accel_mss,speed_ms,0,blend_radius_m)
    |   movel([0.283121, -1.413846, -2.549007, -0.749536, 1.570796, 1.853917],accel_mss,speed_ms,0,blend_radius_m)
    |   movel([0.283324, -1.413314, -2.549408, -0.749667, 1.570796, 1.854121],accel_mss,speed_ms,0,blend_radius_m)
    |   movel([0.283547, -1.412780, -2.549811, -0.749799, 1.570796, 1.854343],accel_mss,speed_ms,0,blend_radius_m)
    |   movel([0.283785, -1.412245, -2.550213, -0.749931, 1.570796, 1.854581],accel_mss,speed_ms,0,blend_radius_m)
    |   movel([0.284041, -1.411712, -2.550613, -0.750064, 1.570796, 1.854837],accel_mss,speed_ms,0,blend_radius_m)
    |   movel([0.284312, -1.411179, -2.551013, -0.750197, 1.570796, 1.855109],accel_mss,speed_ms,0,blend_radius_m)
    |   movel([0.284603, -1.410646, -2.551413, -0.750330, 1.570796, 1.855399],accel_mss,speed_ms,0,blend_radius_m)
    |   movel([0.284890, -1.410142, -2.551790, -0.750457, 1.570796, 1.855687],accel_mss,speed_ms,0,blend_radius_m)
    |   movel([0.285189, -1.409638, -2.552167, -0.750584, 1.570796, 1.855986],accel_mss,speed_ms,0,blend_radius_m)
    |   movel([0.285499, -1.409137, -2.552541, -0.750710, 1.570796, 1.856296],accel_mss,speed_ms,0,blend_radius_m)
    |   movel([0.285820, -1.408639, -2.552913, -0.750837, 1.570796, 1.856616],accel_mss,speed_ms,0,blend_radius_m)
    |   movel([0.286154, -1.408141, -2.553285, -0.750963, 1.570796, 1.856950],accel_mss,speed_ms,0,blend_radius_m)
    |   movel([0.286465, -1.407695, -2.553617, -0.751077, 1.570796, 1.857261],accel_mss,speed_ms,0,blend_radius_m)
    |   movel([0.286788, -1.407252, -2.553947, -0.751190, 1.570796, 1.857585],accel_mss,speed_ms,0,blend_radius_m)
    |   movel([0.287125, -1.406814, -2.554273, -0.751302, 1.570796, 1.857921],accel_mss,speed_ms,0,blend_radius_m)
    |   movel([0.287473, -1.406380, -2.554595, -0.751414, 1.570796, 1.858269],accel_mss,speed_ms,0,blend_radius_m)
    |   movel([0.287831, -1.405952, -2.554913, -0.751524, 1.570796, 1.858628],accel_mss,speed_ms,0,blend_radius_m)
    |   movel([0.288198, -1.405532, -2.555224, -0.751632, 1.570796, 1.858994],accel_mss,speed_ms,0,blend_radius_m)
    |   movel([0.288577, -1.405120, -2.555530, -0.751739, 1.570796, 1.859373],accel_mss,speed_ms,0,blend_radius_m)
    |   movel([0.288965, -1.404713, -2.555832, -0.751844, 1.570796, 1.859761],accel_mss,speed_ms,0,blend_radius_m)
    |   movel([0.289365, -1.404313, -2.556128, -0.751948, 1.570796, 1.860161],accel_mss,speed_ms,0,blend_radius_m)
    |   movel([0.289772, -1.403920, -2.556418, -0.752050, 1.570796, 1.860568],accel_mss,speed_ms,0,blend_radius_m)
    |   movel([0.290226, -1.403501, -2.556728, -0.752160, 1.570796, 1.861023],accel_mss,speed_ms,0,blend_radius_m)
    |   movel([0.290686, -1.403088, -2.557033, -0.752268, 1.570796, 1.861482],accel_mss,speed_ms,0,blend_radius_m)
    |   movel([0.291155, -1.402682, -2.557333, -0.752374, 1.570796, 1.861951],accel_mss,speed_ms,0,blend_radius_m)
    |   movel([0.291630, -1.402283, -2.557626, -0.752479, 1.570796, 1.862427],accel_mss,speed_ms,0,blend_radius_m)
    |   movel([0.292111, -1.401893, -2.557914, -0.752582, 1.570796, 1.862907],accel_mss,speed_ms,0,blend_radius_m)
    |   movel([0.292598, -1.401510, -2.558196, -0.752683, 1.570796, 1.863394],accel_mss,speed_ms,0,blend_radius_m)
    |   movel([0.293092, -1.401135, -2.558472, -0.752782, 1.570796, 1.863888],accel_mss,speed_ms,0,blend_radius_m)
    |   movel([0.293591, -1.400767, -2.558742, -0.752880, 1.570796, 1.864387],accel_mss,speed_ms,0,blend_radius_m)
    |   movel([0.294094, -1.400408, -2.559006, -0.752975, 1.570796, 1.864890],accel_mss,speed_ms,0,blend_radius_m)
    |   movel([0.294554, -1.400091, -2.559238, -0.753060, 1.570796, 1.865351],accel_mss,speed_ms,0,blend_radius_m)
    |   movel([0.295017, -1.399787, -2.559462, -0.753141, 1.570796, 1.865814],accel_mss,speed_ms,0,blend_radius_m)
    |   movel([0.295488, -1.399494, -2.559676, -0.753219, 1.570796, 1.866285],accel_mss,speed_ms,0,blend_radius_m)
    |   movel([0.295964, -1.399210, -2.559884, -0.753295, 1.570796, 1.866760],accel_mss,speed_ms,0,blend_radius_m)
    |   movel([0.296434, -1.398943, -2.560080, -0.753366, 1.570796, 1.867230],accel_mss,speed_ms,0,blend_radius_m)
    |   movel([0.296912, -1.398686, -2.560268, -0.753435, 1.570796, 1.867708],accel_mss,speed_ms,0,blend_radius_m)
    |   movel([0.297390, -1.398441, -2.560447, -0.753501, 1.570796, 1.868187],accel_mss,speed_ms,0,blend_radius_m)
    |   movel([0.297872, -1.398210, -2.560616, -0.753563, 1.570796, 1.868669],accel_mss,speed_ms,0,blend_radius_m)
    |   movel([0.298398, -1.397969, -2.560792, -0.753628, 1.570796, 1.869194],accel_mss,speed_ms,0,blend_radius_m)
    |   movel([0.298923, -1.397740, -2.560959, -0.753690, 1.570796, 1.869719],accel_mss,speed_ms,0,blend_radius_m)
    |   movel([0.299450, -1.397523, -2.561118, -0.753748, 1.570796, 1.870246],accel_mss,speed_ms,0,blend_radius_m)
    |   movel([0.299980, -1.397314, -2.561270, -0.753805, 1.570796, 1.870776],accel_mss,speed_ms,0,blend_radius_m)
    |   movel([0.300614, -1.397079, -2.561442, -0.753869, 1.570796, 1.871411],accel_mss,speed_ms,0,blend_radius_m)
    |   movel([0.301249, -1.396858, -2.561603, -0.753928, 1.570796, 1.872045],accel_mss,speed_ms,0,blend_radius_m)
    |   movel([0.301536, -1.396768, -2.561668, -0.753953, 1.570796, 1.872333],accel_mss,speed_ms,0,blend_radius_m)
    |   movel([0.301823, -1.396688, -2.561726, -0.753974, 1.570796, 1.872619],accel_mss,speed_ms,0,blend_radius_m)
    |   movel([0.302107, -1.396622, -2.561775, -0.753992, 1.570796, 1.872904],accel_mss,speed_ms,0,blend_radius_m)
    |   movel([0.302431, -1.396560, -2.561820, -0.754009, 1.570796, 1.873228],accel_mss,speed_ms,0,blend_radius_m)
    |   movel([0.302757, -1.396507, -2.561858, -0.754023, 1.570796, 1.873553],accel_mss,speed_ms,0,blend_radius_m)
    |   movel([0.303077, -1.396465, -2.561889, -0.754035, 1.570796, 1.873873],accel_mss,speed_ms,0,blend_radius_m)
    |   movel([0.304031, -1.396363, -2.561964, -0.754063, 1.570796, 1.874827],accel_mss,speed_ms,0,blend_radius_m)
    |   movel([0.304981, -1.396269, -2.562032, -0.754088, 1.570796, 1.875778],accel_mss,speed_ms,0,blend_radius_m)
    |   movel([0.305935, -1.396181, -2.562096, -0.754112, 1.570796, 1.876732],accel_mss,speed_ms,0,blend_radius_m)
    |   movel([0.306883, -1.396104, -2.562152, -0.754133, 1.570796, 1.877679],accel_mss,speed_ms,0,blend_radius_m)
    |   movel([0.307197, -1.396086, -2.562165, -0.754138, 1.570796, 1.877994],accel_mss,speed_ms,0,blend_radius_m)
    |   movel([0.307506, -1.396076, -2.562172, -0.754141, 1.570796, 1.878303],accel_mss,speed_ms,0,blend_radius_m)
    |   movel([0.307811, -1.396080, -2.562169, -0.754140, 1.570796, 1.878607],accel_mss,speed_ms,0,blend_radius_m)
    |   movel([0.308070, -1.396096, -2.562157, -0.754135, 1.570796, 1.878866],accel_mss,speed_ms,0,blend_radius_m)
    |   movel([0.308323, -1.396124, -2.562137, -0.754128, 1.570796, 1.879119],accel_mss,speed_ms,0,blend_radius_m)
    |   movel([0.308569, -1.396166, -2.562107, -0.754116, 1.570796, 1.879365],accel_mss,speed_ms,0,blend_radius_m)
    |   movel([0.309105, -1.396279, -2.562024, -0.754085, 1.570796, 1.879901],accel_mss,speed_ms,0,blend_radius_m)
    |   movel([0.309633, -1.396409, -2.561930, -0.754050, 1.570796, 1.880430],accel_mss,speed_ms,0,blend_radius_m)
    |   movel([0.310064, -1.396530, -2.561841, -0.754017, 1.570796, 1.880860],accel_mss,speed_ms,0,blend_radius_m)
    |   movel([0.310487, -1.396666, -2.561743, -0.753980, 1.570796, 1.881284],accel_mss,speed_ms,0,blend_radius_m)
    |   movel([0.310896, -1.396817, -2.561632, -0.753939, 1.570796, 1.881692],accel_mss,speed_ms,0,blend_radius_m)
    |   movel([0.311296, -1.396981, -2.561513, -0.753895, 1.570796, 1.882092],accel_mss,speed_ms,0,blend_radius_m)
    |   movel([0.311683, -1.397160, -2.561382, -0.753846, 1.570796, 1.882480],accel_mss,speed_ms,0,blend_radius_m)
    |   movel([0.312059, -1.397352, -2.561243, -0.753795, 1.570796, 1.882856],accel_mss,speed_ms,0,blend_radius_m)
    |   movel([0.312421, -1.397560, -2.561091, -0.753738, 1.570796, 1.883217],accel_mss,speed_ms,0,blend_radius_m)
    |   movel([0.312771, -1.397779, -2.560931, -0.753679, 1.570796, 1.883567],accel_mss,speed_ms,0,blend_radius_m)
    |   movel([0.313107, -1.398013, -2.560760, -0.753616, 1.570796, 1.883903],accel_mss,speed_ms,0,blend_radius_m)
    |   movel([0.313432, -1.398259, -2.560580, -0.753550, 1.570796, 1.884228],accel_mss,speed_ms,0,blend_radius_m)
    |   movel([0.313741, -1.398518, -2.560390, -0.753480, 1.570796, 1.884537],accel_mss,speed_ms,0,blend_radius_m)
    |   movel([0.314036, -1.398790, -2.560191, -0.753407, 1.570796, 1.884832],accel_mss,speed_ms,0,blend_radius_m)
    |   movel([0.314348, -1.399103, -2.559962, -0.753323, 1.570796, 1.885144],accel_mss,speed_ms,0,blend_radius_m)
    |   movel([0.314641, -1.399433, -2.559721, -0.753235, 1.570796, 1.885437],accel_mss,speed_ms,0,blend_radius_m)
    |   movel([0.314920, -1.399775, -2.559471, -0.753144, 1.570796, 1.885716],accel_mss,speed_ms,0,blend_radius_m)
    |   movel([0.315178, -1.400131, -2.559209, -0.753049, 1.570796, 1.885974],accel_mss,speed_ms,0,blend_radius_m)
    |   movel([0.315421, -1.400496, -2.558941, -0.752952, 1.570796, 1.886217],accel_mss,speed_ms,0,blend_radius_m)
    |   movel([0.315645, -1.400877, -2.558662, -0.752851, 1.570796, 1.886442],accel_mss,speed_ms,0,blend_radius_m)
    |   movel([0.315851, -1.401269, -2.558373, -0.752747, 1.570796, 1.886648],accel_mss,speed_ms,0,blend_radius_m)
    |   movel([0.316037, -1.401673, -2.558076, -0.752640, 1.570796, 1.886834],accel_mss,speed_ms,0,blend_radius_m)
    |   movel([0.316208, -1.402087, -2.557771, -0.752531, 1.570796, 1.887005],accel_mss,speed_ms,0,blend_radius_m)
    |   movel([0.316357, -1.402511, -2.557458, -0.752419, 1.570796, 1.887154],accel_mss,speed_ms,0,blend_radius_m)
    |   movel([0.316491, -1.402947, -2.557137, -0.752305, 1.570796, 1.887287],accel_mss,speed_ms,0,blend_radius_m)
    |   movel([0.316605, -1.403399, -2.556803, -0.752186, 1.570796, 1.887401],accel_mss,speed_ms,0,blend_radius_m)
    |   movel([0.316701, -1.403861, -2.556462, -0.752066, 1.570796, 1.887498],accel_mss,speed_ms,0,blend_radius_m)
    |   movel([0.316779, -1.404331, -2.556115, -0.751944, 1.570796, 1.887576],accel_mss,speed_ms,0,blend_radius_m)
    |   movel([0.316839, -1.404808, -2.555762, -0.751820, 1.570796, 1.887635],accel_mss,speed_ms,0,blend_radius_m)
    |   movel([0.316877, -1.405295, -2.555401, -0.751693, 1.570796, 1.887673],accel_mss,speed_ms,0,blend_radius_m)
    |   movel([0.316899, -1.405787, -2.555036, -0.751566, 1.570796, 1.887695],accel_mss,speed_ms,0,blend_radius_m)
    |   movel([0.316900, -1.406287, -2.554665, -0.751438, 1.570796, 1.887697],accel_mss,speed_ms,0,blend_radius_m)
    |   movel([0.316884, -1.406792, -2.554289, -0.751308, 1.570796, 1.887680],accel_mss,speed_ms,0,blend_radius_m)
    |   movel([0.316848, -1.407303, -2.553909, -0.751177, 1.570796, 1.887644],accel_mss,speed_ms,0,blend_radius_m)
    |   movel([0.316794, -1.407818, -2.553525, -0.751045, 1.570796, 1.887590],accel_mss,speed_ms,0,blend_radius_m)
    |   movel([0.316720, -1.408340, -2.553137, -0.750913, 1.570796, 1.887516],accel_mss,speed_ms,0,blend_radius_m)
    |   movel([0.316626, -1.408871, -2.552740, -0.750778, 1.570796, 1.887423],accel_mss,speed_ms,0,blend_radius_m)
    |   movel([0.316516, -1.409404, -2.552342, -0.750643, 1.570796, 1.887313],accel_mss,speed_ms,0,blend_radius_m)
    |   movel([0.316386, -1.409944, -2.551938, -0.750507, 1.570796, 1.887183],accel_mss,speed_ms,0,blend_radius_m)
    |   movel([0.316241, -1.410482, -2.551536, -0.750372, 1.570796, 1.887038],accel_mss,speed_ms,0,blend_radius_m)
    |   movel([0.316077, -1.411025, -2.551129, -0.750236, 1.570796, 1.886873],accel_mss,speed_ms,0,blend_radius_m)
    |   movel([0.315894, -1.411567, -2.550722, -0.750100, 1.570796, 1.886690],accel_mss,speed_ms,0,blend_radius_m)
    |   movel([0.315695, -1.412112, -2.550313, -0.749964, 1.570796, 1.886491],accel_mss,speed_ms,0,blend_radius_m)
    |   movel([0.315481, -1.412656, -2.549904, -0.749829, 1.570796, 1.886277],accel_mss,speed_ms,0,blend_radius_m)
    |   movel([0.315246, -1.413201, -2.549494, -0.749695, 1.570796, 1.886043],accel_mss,speed_ms,0,blend_radius_m)
    |   movel([0.314999, -1.413744, -2.549084, -0.749561, 1.570796, 1.885795],accel_mss,speed_ms,0,blend_radius_m)
    |   movel([0.314734, -1.414286, -2.548675, -0.749428, 1.570796, 1.885531],accel_mss,speed_ms,0,blend_radius_m)
    |   movel([0.314459, -1.414814, -2.548277, -0.749298, 1.570796, 1.885255],accel_mss,speed_ms,0,blend_radius_m)
    |   movel([0.314169, -1.415341, -2.547879, -0.749170, 1.570796, 1.884965],accel_mss,speed_ms,0,blend_radius_m)
    |   movel([0.313867, -1.415863, -2.547483, -0.749042, 1.570796, 1.884663],accel_mss,speed_ms,0,blend_radius_m)
    |   movel([0.313547, -1.416385, -2.547088, -0.748916, 1.570796, 1.884343],accel_mss,speed_ms,0,blend_radius_m)
    |   movel([0.313216, -1.416904, -2.546695, -0.748790, 1.570796, 1.884012],accel_mss,speed_ms,0,blend_radius_m)
    |   movel([0.312869, -1.417416, -2.546306, -0.748667, 1.570796, 1.883665],accel_mss,speed_ms,0,blend_radius_m)
    |   movel([0.312509, -1.417928, -2.545917, -0.748544, 1.570796, 1.883305],accel_mss,speed_ms,0,blend_radius_m)
    |   movel([0.312136, -1.418431, -2.545534, -0.748423, 1.570796, 1.882933],accel_mss,speed_ms,0,blend_radius_m)
    |   speed_ms = 0.003
    |   movel([0.312136, -1.405810, -2.539761, -0.766817, 1.570796, 1.882933],accel_mss,speed_ms,0,blend_radius_m)
    |   speed_ms = 0.01
    |   movel([0.312136, -1.381543, -2.527823, -0.803023, 1.570796, 1.882933],accel_mss,speed_ms,0,blend_radius_m)
    |   movel([0.175631, -1.306095, -2.578273, -0.828022, 1.570796, 1.746427],accel_mss,speed_ms,0,blend_radius_m)
    |   movel([0.175631, -1.248773, -2.543911, -0.919705, 1.570796, 1.746427],accel_mss,speed_ms,0,blend_radius_m)
    |   # End of main program
    | end
    | 
    | Machining2()
